// ---- 00_FunctionsBlocks/Beckhoff/DataProcessing/Database/SQLite_CreateDb_V2.TcPOU
PROGRAM SQLite_CreateDb_V2
VAR_INPUT
	IN_ConfigDbActuelle		: ARRAY[0..MAX_CONFIGURATIONS] OF ST_ConfigDB; 
	IN_DbType				: UINT:= 1; // 1:T_DBConfig_SQLite, 2:T_DBConfig_SQLCe
	IN_Dir					: T_MAXSTRING;
	IN_Name					: STRING;
	IN_Start				: BOOL;
	IN_TableName			: STRING;
END_VAR
VAR_IN_OUT
	IN_hDBID         		: UDINT;	
END_VAR
VAR_OUTPUT
	OUT_Error				: BOOL;
	OUT_Busy				: BOOL;
	OUT_Result				: INT;
END_VAR
VAR
	Etape					: UINT;
	
	TrigStart				: R_TRIG;
	RsStart					: RS;
	bCreateTable			: BOOL;
	TrigCreateTable			: R_TRIG;
	RsCreateTable			: RS;
	PLCDBCreateEvt 			: FB_PLCDBCreateEvt(sNetID := '', tTimeout := T#5S);
	SqlLiteConf				: T_DBConfig_SQLite;
	DbFullDirName			: T_MAXSTRING;	
	sExtension				: STRING:= '.db';
	tcMessage    	 		: I_TcMessage;
	
	AX_ColArray				: ARRAY[0..3] OF ST_ColumnInfo;
	
	dBID_Test				: UDINT;
	KK						: UDINT;
	bExisteDeja				: BOOL;	
END_VAR

OUT_Busy := TRUE;
AX_ColArray[0].sName := 'TimeStamp';     	AX_ColArray[0].eType := E_ColumnType.DateTime;   	AX_ColArray[0].nLength := 4;    
AX_ColArray[1].sName := 'TimeStamp_Ms';    	AX_ColArray[1].eType := E_ColumnType.Integer;    	AX_ColArray[1].nLength := 4;
AX_ColArray[2].sName := 'ParentId';   		AX_ColArray[2].eType := E_ColumnType.Integer;   	AX_ColArray[2].nLength := 4;
AX_ColArray[3].sName := 'Value';   			AX_ColArray[3].eType := E_ColumnType.Float;   		AX_ColArray[3].nLength := 8;


IF IN_DbType = 1 THEN
	sExtension := '.db';
ELSIF IN_DbType = 2 THEN
	sExtension := '.sdf';
END_IF

DbFullDirName := Concat(STR1:=Concat(STR1:= IN_Dir, STR2 := IN_Name), STR2 := sExtension);
SqlLiteConf.bAuthentification := FALSE;
SqlLiteConf.sServer := DbFullDirName;

FOR KK := 0 TO MAX_CONFIGURATIONS DO
	IF IN_ConfigDbActuelle[KK].sServer = DbFullDirName THEN
		bExisteDeja := TRUE;
		OUT_Result := -1;
		OUT_Busy := FALSE;
		OUT_Error := FALSE;
		bCreateTable := FALSE;
		IN_hDBID := IN_ConfigDbActuelle[KK].hDBID;
		EXIT;
	END_IF
	IF KK = MAX_CONFIGURATIONS THEN
		bExisteDeja := FALSE;
	END_IF
END_FOR

TrigStart(CLK := IN_Start AND NOT bExisteDeja);
RsStart(SET := TrigStart.Q);
IF RsStart.Q1 THEN
	IF PLCDBCreateEvt.Database(pDatabaseConfig := ADR(SqlLiteConf), cbDatabaseConfig := SIZEOF(SqlLiteConf), bCreateXMLConfig := TRUE, pDBID := ADR(dBID_Test)) THEN
		IF PLCDBCreateEvt.ipTcResult.nEventId = 59 THEN
			OUT_Error := FALSE;
			OUT_Result := -1;
			OUT_Busy := FALSE;	
			TrigStart(CLK := FALSE);
			bCreateTable := FALSE;
			Etape := 0;
			RsCreateTable(RESET1 := TRUE);
			RsCreateTable(RESET1 := FALSE);
		ELSIF PLCDBCreateEvt.bError THEN
			tcMessage := PLCDBCreateEvt.ipTcResult;
			OUT_Error := TRUE;
		ELSE
			Etape := 1;
			IN_hDBID := dBID_Test;
			bCreateTable := TRUE; 
		END_IF
		RsStart(RESET1 := TRUE);
		RsStart(RESET1 := FALSE);
	END_IF
END_IF

TrigCreateTable(CLK := bCreateTable);
RsCreateTable(SET:= TrigCreateTable.Q);

IF RsCreateTable.Q1 AND ETAPE = 1 THEN
	IF PLCDBCreateEvt.Table(hDBID := IN_hDBID, sTableName := IN_TableName,  pTableCfg := ADR(AX_ColArray), cbTableCfg := SIZEOF(AX_ColArray)  ) THEN
		IF PLCDBCreateEvt.bError THEN
			Etape := 255;
			OUT_Error := TRUE;
			OUT_Result := -2;
		ELSE
			IN_Start := FALSE;
			bCreateTable := FALSE;
			Etape := 0;
			OUT_Result := 1;
			RsCreateTable(RESET1 := TRUE);
			RsCreateTable(RESET1 := FALSE);
			TrigStart(CLK := False);
			OUT_Busy := FALSE;	
			OUT_Error := FALSE;
		END_IF
	END_IF
END_IF

IF Etape = 255 THEN
	Etape := 0;
	bCreateTable := FALSE;
	IN_Start := FALSE;
	OUT_Busy := FALSE;	
	RsCreateTable(RESET1 := TRUE);
	RsCreateTable(RESET1 := FALSE);
	
END_IF

END_PROGRAM

// ---- 00_FunctionsBlocks/Beckhoff/DataProcessing/Database/SQLite_DeleteConfDb.TcPOU
PROGRAM SQLite_DeleteConfDb
VAR_INPUT
	IN_DbType				: UINT:= 1; // 1:T_DBConfig_SQLite, 2:T_DBConfig_SQLCe
	IN_hDBID         		: UDINT;
	IN_Start				: BOOL;
	
END_VAR
VAR_OUTPUT
	OUT_Error				: BOOL;
	OUT_Busy				: BOOL;
END_VAR
VAR
	Etape					: UINT;
	
	TrigStart				: R_TRIG;
	RsStart					: RS;
	bDeleteTable			: BOOL;
	TrigDeleteFile			: R_TRIG;
	RsDeleteTable			: RS;
	fbConfigTcDBSrv   		: FB_ConfigTcDBSrvEvt (sNetID := '', tTimeout := T#5S);
	DbFullDirName			: T_MAXSTRING;	
	sExtension				: STRING:= '.db';
	tcMessage    	 		: I_TcMessage;
	
	

END_VAR

OUT_Busy := TRUE;

TrigStart(CLK := IN_Start);
RsStart(SET := TrigStart.Q);
IF RsStart.Q1 THEN
	IF fbConfigTcDBSrv.Delete(eTcDBSrvConfigType := E_TcDBSrvConfigType.Database, hConfigID := IN_hDBID) THEN
		IF fbConfigTcDBSrv.bError THEN
			tcMessage := fbConfigTcDBSrv.ipTcResult;
			OUT_Error := TRUE;
			OUT_Busy := FALSE;
			Etape := 255;
		ELSE 
			OUT_Busy := FALSE;
			OUT_Error := FALSE;
			Etape := 0;
		END_IF
		TrigStart(CLK := FALSE);
		RsStart(RESET1 := TRUE);
		RsStart(RESET1 := FALSE);
	END_IF
END_IF

IF Etape = 255 THEN
	Etape := 0;
	bDeleteTable := FALSE;
	IN_Start := FALSE;
	OUT_Busy := FALSE;	
	RsDeleteTable(RESET1 := TRUE);
	RsDeleteTable(RESET1 := FALSE);
	
END_IF

END_PROGRAM

// ---- 00_FunctionsBlocks/Beckhoff/DataProcessing/FB_MessageDynamique.TcPOU
FUNCTION_BLOCK FB_MessageDynamique
// Allows to create dynamic messages in order to add variable to a string
VAR_INPUT
	
	InMessage	: ST_ValuesAlarms;
	InNbparam	: SINT;
END_VAR
VAR_OUTPUT
	OutMessage	: STRING(150);
END_VAR
VAR
	Valeur  	: STRING(10); // Nom de la balise a tester
	P	    	: INT;		 // Pos de la balise dans une chaine de caractere 
	i,j			: SINT;		// Compteur incrémental
	Temp		: String(150);
END_VAR

Temp:=InMessage.Message;
FOR i:=1 TO InNbparam DO
	IF InMessage.Ax_ParamB[i]<>0 THEN
		Valeur := BOOL_TO_STRING(InMessage.Ax_ParamB[i]^);
		P      := FIND(Temp,concat('<Balise_B',INT_TO_STRING(i)));
		IF P >0 THEN
			Temp:=Replace(Temp,Valeur,10,P);
		ELSE
			EXIT;
		END_IF
	END_IF
END_FOR

FOR j:=1 TO InNbparam DO
	IF InMessage.Ax_ParamI[j]<>0 THEN
		Valeur := SINT_TO_STRING(InMessage.Ax_ParamI[j]^);
		P      := FIND(temp,concat('<Balise_I',INT_TO_STRING(j)));
		IF P >0 THEN
			Temp:=Replace(temp,Valeur,10,P);
		ELSE
			EXIT;
		END_IF
	END_IF
END_FOR
OutMessage:=Temp;

END_FUNCTION_BLOCK

// ---- 00_FunctionsBlocks/Beckhoff/DataProcessing/FUN_Transpose.TcPOU
PROGRAM FUN_Transpose
// Allows to transpose an array 
VAR_INPUT
	In_Array					: ARRAY[1..500] OF ARRAY[1..5] OF STRING;
END_VAR
VAR_OUTPUT
	Out_Array					: ARRAY[1..5] OF ARRAY[1..500] OF STRING;
END_VAR


VAR
	KK: INT;
	LL: INT;
END_VAR

FOR LL := 1 TO 5 DO 
	FOR KK := 1 TO 500 DO
	
		Out_Array[LL][KK] := In_Array[KK][LL];
		
	END_FOR
END_FOR

END_PROGRAM

// ---- 00_FunctionsBlocks/Beckhoff/DataProcessing/ReadFile/FB_ReadCSV.TcPOU
FUNCTION_BLOCK FB_ReadCSV
//Permet de lire les Valeurs de max 1 semaine de points (1 pt/min pdt 7 jours)

VAR_INPUT
	InDirectory_Stockage 		: T_MaxString;		// Base file of the Historization 
	InVariable					: T_MaxString;
	InStartTimeStamp			: TIMESTRUCT;
	InNbLecture					: UINT := 144;
	InExecute					: BOOL;			//Rising Edge detection of read
	ParamSeparateur				: STRING;
	InStructValues				: ARRAY[1..500] OF ST_ValuesWrite;
END_VAR                 		

VAR_OUTPUT              		
	OutValue					: ARRAY[1..10000] OF REAL;
	OutTimeStamp				: ARRAY[1..10000] OF TIMESTRUCT;
	OutCompleted				: BOOL;
	OutbBusy					: BOOL;
	OutError 					: BOOL;
	OutErrorID 					: UINT; // 1 : File not found
END_VAR                 		
VAR     
	// Initialisation 
	CP_READ						: BOOL;
	TypeFile					: STRING;
	ParamTimeOut				: TIME := T#1S;
	
	//Read
	TimeStructBeingRead			: TIMESTRUCT;
	FullDirectory				: STRING;                		
	ReadNewFile					: BOOL;
	
	
	OpenFile					: FB_FileOpen;
	ReadFile					: FB_FileGets;
	CloseFile					: FB_FileClose;
	LineStart					: UINT;			// Ligne de début de la lecture
	LineEnd						: UINT;			// Ligne de fin de la lecture
	LineLeft					: UINT;			// Nombre total de lignes restantes
	Index_Array_OutValue		: UINT;			// Valeur de OutValue qui va être écrite
	
	Opening						: BOOL := TRUE;
	Reading						: BOOL;
	Closing						: BOOL;
	LineRead					: ARRAY[1..20] OF T_Maxstring;
	LineReadNull				: ARRAY[1..20] OF T_Maxstring;
	ColumnNbRead				: UINT;
	TimeStampRead				: STRING(255);
	ValueRead					: STRING(255);
	EOF_Reached					: BOOL;
	PosCursor					: DINT;
                    		
	CompteurLigne				: CTU;
	CompteurLigneRead			: CTU;
	OutBusy						: RS;
	Trig_Read					: R_TRIG;
	Trig_Start 					: R_TRIG;
	
	FileHandle					: UINT;
	FileHandle_Old				: UINT;
	
	NbJours						: UINT;
	KK: UINT 					:= 1;
	bInit 						: BOOL;
	FinalElemStruct				: UINT := 20;
	LL							: UINT := 1;
	LenLineRead					: INT;
END_VAR

IF  Trig_Start.Q THEN
	M_Init();
END_IF

CP_Read := SYSTEMTIME_TO_DT(InStartTimeStamp) + LINT_TO_TIME(InNbLecture*60000) < SYSTEMTIME_TO_DT(CalLocalTimeStruct);
 Trig_Start(CLK := InExecute);
CompteurLigneRead(PV := InNbLecture, RESET := Trig_Start.Q);

OutBusy(Set := CP_Read AND InExecute, RESET1 := OutError OR OutCompleted);
OutbBusy := OutBusy.Q1;

OutCompleted := CompteurLigneRead.Q;

IF OutBusy.Q1 THEN	
	// J'initialise le tout : 
		//Initialisation du type de fichier
			TypeFile := 'RAWDATA'; 
			
		// Calcul du nb de fichiers à ouvrir
			NbJours := DINT_TO_UINT( TRUNC(UINT_TO_INT(InNbLecture + InStartTimeStamp.wHour *60 + InStartTimeStamp.wMinute)/(24*60))+1);

	IF KK <= NbJours THEN
		// Nbre d'heures * 60 + Nbre de minutes + 2 lignes de presentation
		IF KK = 1 THEN
			LineStart := (InStartTimeStamp.wHour *60 + InStartTimeStamp.wMinute + 2); 
			// Calcul des lignes de la lecture : 
			LineLeft := InNbLecture;
		ELSE
			LineStart := 2;
		END_IF
		
		LineEnd := MIN(1442, LineLeft);

		CompteurLigne(PV := LineStart+LineEnd);
		
		TimeStructBeingRead := DT_TO_SYSTEMTIME(SYSTEMTIME_TO_DT(InStartTimeStamp) + LINT_TO_TIME(24*3600000*(KK-1)));
		FullDirectory := Concat(Concat(Concat(Concat(Concat(Concat(Concat(Concat(Concat(Concat(Concat(Concat(InDirectory_Stockage , WORD_TO_STRING(TimeStructBeingRead.wyear)),'\'),WORD_TO_STRING(TimeStructBeingRead.wMonth)),'\'),'RAWDATA'),'_'),WORD_TO_STRING(TimeStructBeingRead.wyear)),'-'),WORD_TO_STRING(TimeStructBeingRead.wMonth)),'-'),WORD_TO_STRING(TimeStructBeingRead.wDay)),'.csv');

		//Ouverture du Fichier, récupération du handle
		OpenFile
		(
			sNetId := '',
			sPathName := FullDirectory,
			nMode := FOPEN_MODEREAD,
			ePath := PATH_GENERIC,
			bExecute := Opening AND NOT OutCompleted,
			hFile => FileHandle
		);
		
		IF OpenFile.nErrId = 1804 THEN // Le fichier n'existe pas 
			OutErrorID := 1;
			OutError := OpenFile.bError;
		ELSIF OpenFile.bError THEN		// Il y a eu une autre erreur
			OutError := OpenFile.bError;
		ELSIF NOT OpenFile.bError AND NOT OpenFile.bBusy AND FileHandle <> 0 AND FileHandle <> FileHandle_Old THEN
			Opening := FALSE;
			FileHandle_Old := FileHandle;
		END_IF
		// On a obtenu le file handle, on va commencer la lecture
		
		
		// Le bloc suivant va lire le document ligne à ligne en incrémentant le compteur ligne et en ressortant l'ensemble de la ligne dans LineRead
		
		IF NOT opening AND NOT CompteurLigneRead.Q AND NOT EOF_Reached THEN		
			IF LL <= 20 THEN
				ReadFile
				(
					sNetId := '',
					hFile := FileHandle,
					bExecute := TRUE,
					tTimeout := ParamTimeOut,
					sLine => LineRead[LL],
					bEOF => EOF_Reached
				);	
				IF NOT ReadFile.bBusy AND NOT ReadFile.bError AND lineread[LL] <> '' THEN
					ReadFile(bExecute := FALSE);
					LenLineRead := LEN(STR := LineRead[LL]);
					IF LenLineRead = 254 THEN
						LL := LL + 1 ;
					ELSE
						FinalElemStruct := LL;
						LL := 1;
					END_IF
				END_IF
			END_IF
			
			IF NOT ReadFile.bBusy AND NOT ReadFile.bError AND (LineRead[FinalElemStruct] <> '' OR EOF_Reached) THEN
				ReadFile(bExecute := FALSE);
				CompteurLigne(CU := TRUE);	
				CompteurLigne(CU := FALSE);
				FinalElemStruct := 20;
				
				IF CompteurLigne.CV >= LineStart + 1 THEN
					TimeStampRead := Substring_Cari
					(
						IN_Delimiter := ParamSeparateur, 
						IN_TextToSearch := LineRead, 
						IN_Position := 0
					);
					OutTimeStamp[Index_Array_OutValue+1]:= FUN_FormatDate(In_String := TimeStampRead);
					
					ValueRead := Substring_Cari
					(
						IN_Delimiter := ParamSeparateur, 
						IN_TextToSearch := LineRead, 
						IN_Position := ColumnNbRead + 1
					);
					OutValue[Index_Array_OutValue+1] := STRING_TO_REAL(ValueRead)*100;
					CompteurLigneRead(CU := TRUE);
					CompteurLigneRead(CU := FALSE);
					Index_Array_OutValue := Index_Array_OutValue + 1;
					
					LL := 1;
				END_IF
				LineRead := LineReadNull;
			ELSIF NOT ReadFile.bBusy AND  ReadFile.bError THEN
				OutError := TRUE;			
			END_IF
		ELSIF EOF_Reached THEN
			ReadFile(bExecute := FALSE);
	
			CloseFile
			(
				sNetId := '',
				bExecute := TRUE,
				hFile := FileHandle,
				tTimeout := ParamTimeOut
			);
			IF NOT CloseFile.bBusy AND NOT CloseFile.bError  THEN
				LineLeft := LineLeft - CompteurLigneRead.CV + 2;
				Index_Array_OutValue := Index_Array_OutValue -1;
				CloseFile(bExecute := FALSE);
				CompteurLigne(RESET := TRUE);
				CompteurLigne(RESET := FALSE);
				Opening := TRUE;
				EOF_Reached := FALSE;
				KK := KK + 1;
			END_IF	
		END_IF
	END_IF
ELSIF EOF_Reached OR CompteurLigneRead.Q AND FileHandle <> 0 THEN
	ReadFile(bExecute := FALSE);
	
	CloseFile
	(
		sNetId := '',
		bExecute := TRUE,
		hFile := FileHandle,
		tTimeout := ParamTimeOut
	);
	IF NOT CloseFile.bBusy AND NOT CloseFile.bError THEN
		CloseFile(bExecute := FALSE);
		CompteurLigne(RESET := TRUE);
		CompteurLigne(RESET := FALSE);
		Opening := TRUE;
		Index_Array_OutValue := 0;
		FileHandle := 0;
		KK := 1;
	ELSIF NOT CloseFile.bBusy AND closefile.bError THEN
		OutError := TRUE;
	END_IF  
END_IF

METHOD M_Init : BOOL
VAR_INPUT
END_VAR

VAR
	KK : UINT;
END_VAR
ColumnNbRead := 1;
FOR KK := 1 TO 500 DO
	IF InVariable = InStructValues[KK].Description THEN
		ColumnNbRead := KK;
		EXIT;
	END_IF
END_FOR
END_METHOD

END_FUNCTION_BLOCK

// ---- 00_FunctionsBlocks/Beckhoff/DataProcessing/WriteFile/CheckStruct_Alarms.TcPOU
FUNCTION CheckStruct_Alarms : BOOL
//Allows to compare 2 Struct_InputRTU, TRUE if struct are the same
VAR_INPUT
	InStruct1 : ST_ValuesAlarms;
	InStruct2 : ST_ValuesAlarms;
END_VAR
VAR
	bCompareBuffer 	: BOOL := TRUE;
	KK 				: UINT;
END_VAR

CheckStruct_Alarms := InStruct1.Message = Instruct1.Message and InStruct1.ID = Instruct2.ID and InStruct1.Value = InStruct2.Value and InStruct1.Written = Instruct2.Written;

END_FUNCTION

// ---- 00_FunctionsBlocks/Beckhoff/Fifo/FB_CommandAlternate.TcPOU
FUNCTION_BLOCK FB_CommandAlternate
VAR_INPUT
	AX_CMD 			: ARRAY[1..6] OF INV_Cmd;
	In_NB_Prio		: UINT;							
	ParamNbCMD		: UINT := 6;					// Number of elements of AX_CMD array
	In_Pulse		: BOOL;
END_VAR

VAR_OUTPUT
	CmdOutput		: INV_Cmd	;
END_VAR
VAR
	LastPosition 	: UINT;
	KK				: UINT;
	bInterrupt		: BOOL;
	Debut			: UINT;
	Fin				: UINT;
	Trig_Detec		: R_TRIG;
END_VAR

bInterrupt := FALSE;
Trig_Detec(CLK := In_Pulse);

IF Trig_Detec.Q THEN
	FOR KK := 1 TO In_NB_Prio DO
		IF AX_CMD[KK].bCmdStart^ THEN
			bInterrupt 	:= TRUE;
			CmdOutput := AX_CMD[KK];
			EXIT;
		END_IF
	END_FOR
	
	IF NOT bInterrupt THEN
		Debut := MAX(In_NB_Prio + 1, LastPosition + 1);
		Fin := Debut + ParamNbCMD - In_NB_Prio - 1;
		FOR KK := Debut TO Fin DO
			IF AX_CMD[KK - BOOL_TO_UINT(KK > ParamNbCMD)*(Fin - Debut + 1)].bCmdStart^ THEN
				LastPosition := KK - BOOL_TO_UINT(KK > ParamNbCMD)*(Fin - Debut + 1);
				CmdOutput := AX_CMD[ KK - BOOL_TO_UINT(KK > ParamNbCMD)*(Fin - Debut + 1)];
				EXIT ;
			END_IF
		END_FOR
	END_IF
END_IF

END_FUNCTION_BLOCK

// ---- 00_FunctionsBlocks/Common/AlarmManagement/FB_DetectFixedValue.TcPOU
FUNCTION_BLOCK FB_DetectFixedValue
VAR_INPUT
	IN_Addr			: POINTER TO BYTE;			// Adr of the variable to  analyse
	IN_EmptyStruct	: POINTER TO BYTE;			// Adr of a null variable on which I input the compared value
	IN_Size			: UINT;						// Size of the variable to analyse
	IN_Duration		: TIME;						// Duration after which an alarm is raised
END_VAR
VAR_OUTPUT
	OUT_bStatic		: BOOL;						// Value has been static for more than IN_Duration time
END_VAR
VAR
	TON_CMP			: TON;
	bFixed			: BOOL;
END_VAR

bFixed :=  MEMCMP(pBuf1 := IN_Addr, pBuf2 := IN_EmptyStruct, n := IN_SIZE)=0;

TON_CMP(IN := bFixed, PT := IN_Duration, Q => OUT_bStatic);

IF NOT bFixed THEN
	MEMCPY(destAddr := IN_EmptyStruct, srcAddr := IN_Addr, n := IN_Size);
END_IF

END_FUNCTION_BLOCK

// ---- 00_FunctionsBlocks/Common/AlarmManagement/FB_UnknownEvent.TcPOU
FUNCTION_BLOCK FB_UnknownEvent
////////////////// 
// Detect an event that is not the result of an internal command, or an external event
//////////////////	
VAR_INPUT
	IN_TempoAfterCommand					: TIME ;					// Tempo between internal command and event
	IN_TempoReadExternalEvent					: TIME ;					// Tempo to read the external event
	
	IN_InternalCommand				: BOOL ; 			// Internal command that normally trigers the event 
	IN_ExternalEvent				: BOOL ; 			// External Event that normally explains the Event (to be read after the event)
	
	IN_Event						: BOOL ; // Event that occur
	
	bReset				: BOOL := FALSE ; 	// Reset 
	
END_VAR

VAR_OUTPUT
	OUT_Unknown 			: BOOL ; 		// Flag to TRUE is the event is unknown ( neither related to the command, or an external event that is known) 
	
END_VAR

VAR
	FB_CheckCommand : FB_CheckCommand ;
	// Inconsistency detection
	R_TRIG1				: R_TRIG ; 		// Detect command
	TOF1				: TOF ; 		// Creates a falling edge T time after command detcetion	
	F_TRIG				: F_TRIG ; 		// Detect Falling edge of TOF1	
	
	F_TRIG2				: F_TRIG ; 		// Detect falling edge of feedback measure
	TOF2				: TOF ; 		// Creates  a falling edge T time after Feedback measure ended detcetion
 
	TON					: TON ; 		// Tempo in case of bistable functuion

	// Reset management 	
	TOF_Reset			: TOF;			// Hold Reset command afetr reset to inhibate future warnings
	RS_Reset			: RS;			// Maintain reset command
	
	R_TRIG2: R_TRIG;
	CalNotLinkedToCommand: BOOL;
END_VAR


R_TRIG1(CLK := IN_InternalCommand) ; 

TOF1(IN:=R_TRIG1.Q , PT:=IN_TempoAfterCommand) ;
F_TRIG(CLK:=TOF1.Q);		

R_TRIG2(CLK := IN_Event) ; 


CalNotLinkedToCommand :=  NOT TOF1.Q AND R_TRIG2.Q ;
 
FB_CheckCommand(T:= IN_TempoReadExternalEvent , bCmd := CalNotLinkedToCommand , bMes := IN_ExternalEvent , bReset := bReset , bImpulsion := TRUE ) ; 
OUT_Unknown := FB_CheckCommAND.bWarning  ;

END_FUNCTION_BLOCK

// ---- 00_FunctionsBlocks/Common/BoolManagement/FB_CountNinTimeWindow.TcPOU
FUNCTION_BLOCK FB_CountNinTimeWindow
VAR_INPUT
	IN_CountMax			: UINT := 3 ; 
	IN_bInput				: BOOL;
	IN_bReset			: BOOL;
END_VAR
VAR_OUTPUT
	OUT_FlagNinT		: BOOL;		// Output : if CountMax Input occured in the last T min, this variable = TRUE;
END_VAR
VAR
	TimeFault1			: TIME;		// Temps du troisième défaut GTE (chronologiquement parlant)
	TimeFault2			: TIME;		// Temps du deuxième défaut GTE (chronologiquement parlant)
	TimeFault3			: TIME;		// Temps du premier défaut GTE (chronologiquement parlant)
	TriggerGTE			: R_TRIG;	
	
	TestDiff			: TIME;
END_VAR
VAR_INPUT PERSISTENT
	ParamTimeToMeasure	: TIME := T#30M; // Time during which the 3 GTE are measured. Used for testing.
END_VAR

TriggerGTE(CLK:= IN_bInput);

 IF IN_bReset THEN
		OUT_FlagNinT := FALSE;
		TimeFault1 := T#0S;
		TimeFault2 := T#0S;
		TimeFault3 := T#0S;
END_IF

IF TriggerGTE.Q AND TimeFault3 = T#0S THEN
	TimeFault3 := TIME();
ELSIF TriggerGTE.Q AND TimeFault2 = T#0S THEN
	TimeFault2 := TIME();
ELSIF TriggerGTE.Q AND TimeFault1 = T#0S THEN
	TimeFault1 := TIME();
ELSIF TriggerGTE.Q THEN
	TimeFault3 := TimeFault2;
	TimeFault2 := TimeFault1;
	TImeFault1 := TIME();
END_IF


IF TimeFault1 - TimeFault3 < ParamTimeToMeasure AND TimeFault1 <> T#0S THEN
	OUT_FlagNinT := TRUE;
ELSE 
	OUT_FlagNinT := FALSE;
END_IF

END_FUNCTION_BLOCK

// ---- 00_FunctionsBlocks/Common/BoolManagement/FB_Toggle2Tap.TcPOU
FUNCTION_BLOCK FB_Toggle2Tap
///////////
// FB to change a toggle into a tap with constant duration//
///////////

VAR_INPUT
	TapDuration		: TIME; 	// (s) Tap duration
	
	ToggleVar 		: BOOL;		// Toggled input variable 

	
END_VAR

VAR_OUTPUT
	TapVar			: BOOL ; 	// Tapped output variable
	
END_VAR

VAR				
	R_TRIG			: R_TRIG ;				// Create a square at Rising Edge Detection
	F_TRIG			: F_TRIG ;				// Create a square at falling Edge Detection 
	TP				: TP ; 					// Square Signal 

END_VAR

R_TRIG(CLK := ToggleVar) ;  							// Rising Edge Detection
F_TRIG(CLK := ToggleVar) ; 								// Falling Edge Detection

TP(IN := R_TRIG.Q OR F_TRIG.Q , PT := TapDuration) ;  	// Square signal 

TapVar		:= TP.Q ; 									// OUtput variable

END_FUNCTION_BLOCK

// ---- 00_FunctionsBlocks/Common/BoolManagement/FB_WriteOnChange.TcPOU
FUNCTION_BLOCK FB_WriteOnChange
////////////////// 
// Write output variable , equals to input variable only if input variable changed state 
//////////////////	

VAR_INPUT
	Size			: UDINT; 				// Variable size 
	VarOut			: POINTER TO BYTE;		// Output  Variable Memory Address
	VarInput		: POINTER TO BYTE;		// Input Variable Memory Address	
END_VAR


VAR
	VarHold 		: DWORD  ; 	

END_VAR

IF MEMCMP(pBuf1:= VarInput, pBuf2:= ADR(VarHold) , n:=Size )<>0  THEN
	MEMCPY(srcAddr:= VarInput , destAddr := VarOut, n:= Size ) ;
END_IF

IF MEMCMP(pBuf1:= VarOut, pBuf2:= ADR(VarHold) , n:=Size )<>0  THEN
	MEMCPY(srcAddr:= VarOut , destAddr := VarInput, n:= Size ) ;
END_IF

MEMCPY(srcAddr:= VarInput , destAddr := ADR(VarHold), n:= Size ) ;

END_FUNCTION_BLOCK

// ---- 00_FunctionsBlocks/Common/BoolManagement/RS_NoReset.TcPOU
FUNCTION_BLOCK RS_NoReset
//Output reset the input if the input is false 
VAR_INPUT
	Set 		: BOOL;
	Reset 		: BOOL;
END_VAR
VAR_OUTPUT
	Q1 			: BOOL;
END_VAR
VAR
	TRIG 		: R_TRIG;
	RS 			: RS;
END_VAR

TRIG(CLK := Set);
RS(Set := TRIG.Q, RESET1 := Reset AND NOT Set, Q1 => Q1);

END_FUNCTION_BLOCK

// ---- 00_FunctionsBlocks/Common/Ctrl/FB_PIDRegulation.TcPOU
FUNCTION_BLOCK FB_PIDRegulation
// Akuo Version of PID Regulation  for solar power plant . Input can be P or Q . 
// Out  = Error *K (1+ 1/Ti sum(error) + Td delta(error) ) 
(*
	DATE :						07/2020																										
	Developper:				GGY																												
	Version :					V1.0																										
	Function :																																																																		
*)
VAR_INPUT PERSISTENT

	ParamK				: REAL ; // Proportionnal 
	ParamTi				: REAL ; // Integral (s) . 0 to disable
	ParamTd				: REAL ; // Derivative (s). 0 to disable . 
	
	ParamXmax			: REAL ; // maximal Value for X. Shall account for number of available PTR . 
	ParamXmin			: REAL; // minimal value for X 
	
	ParamOutmax			: REAL ; // Maximal output value
	ParamOutmin			: REAL ; // Maximal input value 
	
	
	
END_VAR

VAR_INPUT
	IN_SetptX				: REAL ; // Value to reach 
	IN_MesX					: REAL ; // Measure to compare with
	IN_MesComXError			: BOOL ; // Communication lost with the measure tool. 
	IN_SetptOpenLoop		: REAL  ; // Output of the PID when disabled. This shall be equal to an evaluation of the correct output. Usually SetptX. OpenLoop setpoint. 

	
	IN_CmdReset				: BOOL ; // Reset PID 
	IN_CmdPIDOn				: BOOL ; // Activate/ Desactivate PID . outpout equals to the offset if desactivated/ 
END_VAR

VAR_OUTPUT
	OUT_X					: REAL ; // Output of the PID 
	OUT_PIDMode				: INT ; // Mode of the PID ( 1: Bypassed  , 3 : Proportionnal , 4 : PI , 5 PID , 6: PD). 
	
END_VAR
VAR
	
	CalSetptOffset 			: REAL  ; // Offset to be added to the PID to ensure continuity when resetting it or activating it. 

	IntegralX			: REAL ; // Intergal
	DerivativeX			: REAL ; // Derivative
	ErrorX				: REAL;	// Error  
	CP_PID				: BOOL;	// PID Enabled
	Clock				: TON ; // Calculate Elapsed Time ; 
	DeltaTime			: REAL ; // 
	// Derivative
	StepDerivative		: INT := 0; // Derivative Step ( initialization , methode degre 1 , methode degre 2) 
	X2,X1				:REAL;
	T1					:REAL;
	CalReset: BOOL;
	
	KCopy				: REAL ; 
	TiCopy				: REAL ; 
	TdCopy				: REAL ; 
	X_Temp				: REAL ; // Intermediate result . 
	
	CalOutLimitReached_Up	: BOOL;		// Output reached maximum output limit
	CalOutLimitReached_Down	: BOOL;		// Output reached minimum output limit
	
	TrigCP_PID: BOOL;
	bInit: BOOL := TRUE  ; 
	time_new: INT;
	delta_time: INT;
	time_old: INT;
END_VAR

// INITIALIZE 
	OUT_PIDMode := 1 ;

	CalReset := IN_CmdReset OR NOT IN_CmdPIDOn OR ABS(KCopy-ParamK)>0.000001 OR ABS(TiCopy-ParamTi)>0.000001 OR ABS(TdCopy-ParamTd)>0.000001 OR IN_MesComXError; // Reset if change of parameters >> passage en boucle ouverte. 

	CP_PID :=   (ParamK>0.00001 OR ParamK<-0.00001)  AND NOT CalReset  ; // PID Enable ssi Activation and K >0 and not communication alarm with power meter . and not K change . 
	

	IF NOT CP_PID OR bInit THEN 
		// Début proposition de modif KBT
		time_old := TIME_TO_INT(TIME());
		// Fin proposition de modif KBT

		
		Clock(IN:=FALSE ) ; 
		Clock(IN:=TRUE, PT:=T#1H);	//Initialize clock 
		bInit	:= FALSE ; 
	ELSE 
		Clock();
		DeltaTime	:= TIME_TO_REAL(CLOCK.ET)/1000 ; 	// in seconds
		
		// Début proposition de modif KBT
		time_new := TIME_TO_INT(TIME());
		IF time_old <> 0 THEN
			delta_time := time_new - time_old;
		END_IF
		time_old := TIME_TO_INT(TIME());
		// Fin proposition de modif KBT
	END_IF


	KCopy 	:=  ParamK ; 
	TiCopy	:= ParamTi ; 
	TdCopy	:= ParamTd ; 
	
// CHECK INPUT // 
	IN_SetptX := MAX(MIN(IN_SetptX, ParamXmax ), ParamXmin); // Limit the Input with Min/ Max values.

	IN_SetptOpenLoop := MAX(MIN(IN_SetptOpenLoop, ParamXmax ), ParamXmin); // Limit the Input with Min/ Max values.
	
// EVALUATE QUANTITIES //
	// Clock
	
	IF DeltaTime > 0 THEN	// We calculate on time cycle. When the time cycle is over , we reinitialize the clock
		Clock(IN:=FALSE ) ; 
		Clock(IN:=TRUE, PT:=T#1H);	//Initialize clock 
	ELSE
		CLOCK(PT:=T#1H,IN:=TRUE);
	END_IF
	// Error 
		ErrorX := IN_SetptX - IN_MesX ; 

	//Integral
		// Sauturate the integral if overflow or if limts are reached or output reaches limits Reset the integral if command reset. 
		IF (NOT(1E30 - ErrorX*DeltaTime < IntegralX OR -1E30 - ErrorX*DeltaTime > IntegralX) AND ParamTi>0 ) OR CalReset THEN
			IF NOT ((ErrorX > 0 AND  CalOutLimitReached_Up) OR (ErrorX < 0 AND CalOutLimitReached_Down)) THEN 
				IntegralX:=SEL(CalReset,IntegralX+ErrorX*DeltaTime , 0) ;
			END_IF
			
			
		END_IF
		
	// Derivative 
		IF StepDerivative=0 OR CalReset THEN		// Reinitializa derivative if reset commAND  
			X1:=ErrorX;
			X2:=ErrorX;
			T1:=DeltaTime;
			DerivativeX := 0;
			StepDerivative:=1;
		ELSIF StepDerivative=1 AND ParamTd>0 THEN 
			DerivativeX := (ErrorX - X1)/(DeltaTime-T1) ; // f'(x) = (f(x+h)-f(x))/h
			X2:=X1;
			X1:=ErrorX;
			T1:=DeltaTime;	
			StepDerivative:=2 ; 		
		ELSE	
			IF DeltaTime>0 AND DerivativeX < 1E30 AND ParamTd>0  THEN		// Saturate the derivative if going too high. 
				IF NOT ((ErrorX > 0 AND  CalOutLimitReached_Up) OR (ErrorX < 0 AND CalOutLimitReached_Down)) THEN  
					DerivativeX:=(3*(ErrorX)-4*X1+X2)/(2*(DeltaTime-T1));		// Formule de Gear au second degré décentré à gauche . f'(x) = 1/2h*(3*f(x+2h)-4*f(x+h)+f(x))  >>> https://www.imo.universite-paris-saclay.fr/~francois.dubois/cours/iacs/iacs-chap05.pdf
					X2:=X1;
					X1:=ErrorX;
					T1:=DeltaTime;
				END_IF
			END_IF;
		END_IF;
	
// PID CALCULATION
	IF CP_PID THEN

		
		TrigCP_PID	:= TRUE ; 
		// PID Enable 
		IF  ParamTi>0 AND ParamTd>0 THEN // Integral and derivative activated
			X_Temp:=CalSetptOffset+ParamK*(ErrorX+IntegralX/ParamTi+DerivativeX*ParamTd);
			OUT_PIDMode := 5 ; 
		ELSIF ParamTd>0 THEN // Derivative activated 
			X_Temp:= CalSetptOffset+ParamK*(ErrorX+DerivativeX*ParamTd) ; 
			OUT_PIDMode := 6 ; 
		ELSIF ParamTi>0 THEN // Integral activated 
			X_Temp:=CalSetptOffset+ParamK*(ErrorX+IntegralX/ParamTi);
			OUT_PIDMode := 4 ; 
		ELSE	// Only proportionnal
			X_Temp:=CalSetptOffset+ParamK*(ErrorX) ; 
			OUT_PIDMode := 3 ; 
		END_IF
		
	ELSE
		
		CalSetptOffset := IN_SetptOpenLoop ; // At the moment when i activated the PID, i need to ensure continuity of the OUT_X and start the PID from there . 
	
		TrigCP_PID	:= FALSE ; 
		//PID Disable. Open Loop . 
		X_Temp := IN_SetptOpenLoop ;
		OUT_PIDMode:=1 ;
	END_IF
	
// Saturate the OUtput with limits : 
CalOutLimitReached_Up := (X_Temp > ParamOutmax)  ;
CalOutLimitReached_Down:= (X_Temp < ParamOutmin)  ;
 

OUT_X :=  MAX(MIN(ParamOutmax , X_Temp ) , ParamOutmin ) ;

END_FUNCTION_BLOCK

// ---- 00_FunctionsBlocks/Common/DataProcessing/FB_CountBitOfWordAtTrue.TcPOU
FUNCTION_BLOCK FB_CountBitOfWordAtTrue
// Count the number of active bit of a word
VAR_INPUT
	MyWord		 	: WORD;		
END_VAR
VAR_OUTPUT
	NbrBitAtTrue 	: BYTE;
	PosOfLastOne	: BYTE;
END_VAR
VAR
	KK 			 	: BYTE;
	VarTemp		 	: WORD;
END_VAR


NbrBitAtTrue := 0;
FOR KK := 1 TO 16 DO
	Vartemp := ROL(MyWord, KK);
	IF VARtemp.0 THEN
		NbrBitAtTrue := NbrBitAtTrue +1 ;
		PosOfLastOne := KK;
	END_IF
END_FOR

END_FUNCTION_BLOCK

// ---- 00_FunctionsBlocks/Common/DataProcessing/FB_Integrate.TcPOU
FUNCTION_BLOCK FB_Integrate
// This FB increments the value of the Input with every call of the FB. DO NOT CALL THIS TWICE IN A CYCLE.
// Integration is done with the trapeze method
// The Reset input resets the value to 0
VAR_INPUT
	IN_DataToIntegrate		: REAL;
	IN_CmdReset				: BOOL;
	
END_VAR
VAR_OUTPUT
	OUT_IntegrationValue	: REAL;
END_VAR
VAR
	OldData					: REAL;
	OldTime					: TIME;
	DeltaTime				: TIME;
END_VAR

IF OldTime > T#0S THEN
	DeltaTime := TIME()-OldTime;
	
	OUT_IntegrationValue := OUT_IntegrationValue+(IN_DataToIntegrate + OldData)*TIME_TO_REAL(DeltaTime)/2000.0;
	
	OldTime := TIME();
	OldData := IN_DataToIntegrate;
	
	IF IN_CmdReset THEN
		OUT_IntegrationValue := 0.0;
		OldData := 0.0;
	END_IF
ELSE
	OldTime := TIME();
	OldData := IN_DataToIntegrate;
END_IF

END_FUNCTION_BLOCK

// ---- 00_FunctionsBlocks/Common/DataProcessing/FB_MovingAverage.TcPOU
FUNCTION_BLOCK  FB_MovingAverage
//////////////////
// Calculate the Moving Average of a data. Maximal number of point.
//////////////////

VAR CONSTANT 
	CstNbPointMax			: INT := 1000 ; // Average on one hour, with seconds granularity points

END_VAR


VAR_INPUT
	WindowDuration		: DINT ; // (ms) Window of Time during which the average will be done . 
	ValueIn 			: REAL ; // Value to average
	UpdatePeriod		: DINT ; // (ms) Period at which the value is updated. 	
	CycleTime			: INT := CstCycleTime_G; // (ms) Cycle time of the CPU
END_VAR
	

VAR_OUTPUT
	ValueOut			: REAL ; // Averaged Value. 
	bError 				: BOOL ; // Switch to true if error i inputs				
END_VAR

VAR
	Values 				: ARRAY[1..CstNbPointMax] OF REAL; 	// Value to remove from the average calculation
	
	NbPoints			: DINT ; 	// Number of points used for calculating the average. 
	PointPickUpNb		: DINT ; 	// Number of points to skip in average calculation
	
	JJ					: DINT;		// Pick Up index . 
	KK					: DINT;		// For Loop 
	
END_VAR

// EVALUATE VARIABLES //
PointPickUpNb 	:= UpdatePeriod		/	CycleTime ;
NbPoints 		:= WindowDuration 	/ 	UpdatePeriod  ;  

// CHECK INPUTS //
IF NbPoints > CstNbPointMax THEN 
	bError 		:= TRUE ; 
	ValueOut 	:= -1 ;
	
ELSE
	// UPDATE VALUE ARRAY WITH NEW VALUE AND REMOVE OLD ONE //
	JJ			:=JJ+1 ;
	
	IF JJ = PointPickUpNb THEN 
		JJ		:= 0 ; // Reinitialize JJ
		
		// Move all values in the array on the right
		FOR KK :=1 TO NbPoints-1 DO 
			Values[NbPoints-KK+1]	:= Values[NbPoints-KK] ;
			
		END_FOR
		
		Values[1] 					:= ValueIn ; 	// Assign first index to new value. 
		
		// CALCULATE AVERAGE // 
			ValueOut 						:= 0 ; 
			
			FOR KK:=1 TO NbPoints DO 
				ValueOut 					:= ValueOut + Values[KK] / DINT_TO_REAL(NbPoints) ; 
			
			END_FOR
		
	END_IF
END_IF

END_FUNCTION_BLOCK

// ---- 00_FunctionsBlocks/Common/DataProcessing/FB_Ramp.TcPOU
FUNCTION_BLOCK FB_Ramp
VAR_INPUT
	IN			: REAL;							(* New Setpoint variable *)
	ASCEND		: REAL;					(* maximum positive slope. Set negative value for no limit *)
	
	DESCEND		: REAL;				(* maximum negative slope (non-negative!!).Set negative value for no limit *)
	TIMEBASE	: TIME;					(* reference for ASCEND/DESCEND :
											t#0s : ASCEND/DESCEND defined per call
											else : ASCEND/DESCEND defined per specified time *)
	IN_RESET_VALUE		: REAL; // Value at which the OUT is reseted 
	RESET				:BOOL;						(* reset *)
END_VAR
VAR_OUTPUT
	OUT								: REAL;						(* output limited by  slope *)
	Out_Completed 					: BOOL ; // True when the ramp is over. 
END_VAR
VAR
	DIFF: REAL;
	OLD_IN: REAL;
	TB,CET:DWORD;
	CLOCK: TON;
	probe:REAL;
END_VAR

Out_Completed := FALSE ;

IF RESET=TRUE OR CLOCK.PT<>TIMEBASE THEN			(* Reset *)
	OUT :=  IN_RESET_VALUE ; 
	OLD_IN:=OUT;
	CLOCK(PT:=TIMEBASE,IN:=FALSE);
	Out_Completed := TRUE  ;
END_IF

DIFF:=IN-OLD_IN;									(* Calculate setpoint difference between old and new setpoint *)

IF TIMEBASE=T#0S THEN								(* PLC Cycletime *)
	IF DIFF>ASCEND AND ASCEND >0 THEN
		OUT:=OLD_IN+ASCEND;
	ELSIF DIFF<-DESCEND AND DESCEND >0 THEN
		OUT:=OLD_IN-DESCEND;
	ELSE
		OUT:=IN;
		Out_Completed := TRUE  ;					// 
	END_IF;
ELSE												(* Slope per timebase *)
	TB:=TIME_TO_DWORD(TIMEBASE);					(* TIMEBASE as DWORD *)
		CLOCK();
	CET:=TIME_TO_DWORD(CLOCK.ET);					(* Elapsed time : correspond to cycle time*)
	IF CET>0 THEN									(* *)
		CLOCK(IN:=FALSE);							(* Restart timer *)
		CLOCK(IN:=TRUE);
		probe:=DIFF*TB/CET;							// SMesIng value difference to fit timebase
		IF probe>ASCEND AND ASCEND >0 THEN						(* ascending *)
			OUT:=OLD_IN+ASCEND*CET/DWORD_TO_REAL(TB);
		ELSIF probe<-DESCEND AND DESCEND >0 THEN					(* descending *)
			OUT:=OLD_IN-DESCEND*CET/DWORD_TO_REAL(TB);
		ELSE										(* If value between max descend and max ascend.  *)
			OUT:=IN;
			Out_Completed := TRUE  ;
		END_IF;
	ELSE											(* keine Zeit verstrichen *)
		CLOCK.PT:=TIMEBASE;							(* => ggf. Initialisierung *)
		CLOCK(IN:=TRUE);							(* => ggf. Timer neu starten *)
		Out_Completed := TRUE  ;
	END_IF;
END_IF;

OLD_IN:=OUT;

END_FUNCTION_BLOCK

// ---- 00_FunctionsBlocks/Common/DataProcessing/FB_Ramp_Time.TcPOU
FUNCTION_BLOCK FB_Ramp_Time
// Y := Ax + B while bStart is set
// Works with time : You can set a max time, and a duration of the ramp :
// if pause is True, the Y value freezes until pause goes to False
// if max time is reached, the Y value goes to the value at maxtime

VAR_INPUT
	A 								: REAL ;	// Slope of the ramp
	B 								: REAL ;	// Initial value of the ramp
	bStart 							: BOOL ;	// Rising edge detection to start the ramp, if false, the ramp stops
	bPause							: BOOL ; 	// Pause signal : the value stop, then continues when bPause goes to false
	RampTime						: TIME ;	// Duration of the ramp
	MaxRampTime						: TIME ; 	// Maximum duration of the ramp (including breaks)
END_VAR                 			

VAR_OUTPUT              			
	Y 								: REAL;
	OutCompleted					: BOOL; 	// Rising edge detection to indicate the ramp is done
END_VAR                 		
	
VAR                     			
	TimeStart 						: TIME;
	TimeDurationPause 				: TIME;
	TimeOnGoing						: TIME;
	TimePauseold					: TIME;
	
	Trig_Start						: R_TRIG;
	Trig_Stop						: F_TRIG;
	Trig_PauseStart					: R_TRIG;
    Trig_OutCompleted				: R_TRIG;
            			
	Real_TimeSinceInit 				: REAL;
	                    	
	RS_TimerOn						: RS;
	TP_RampMaxTime					: TP;
END_VAR

Trig_Start(CLK := bStart);
TP_RampMaxTime(IN := Trig_Start.Q, PT := MaxRampTime);


//Trig_Stop(Clk := bStart AND TP_RampMaxTime.Q );
Trig_PauseStart(CLK := bPause);
Trig_OutCompleted(CLK := RS_TimerOn.Q1 AND TimeOnGoing = RampTime);

RS_TimerOn(SET := Trig_Start.Q, RESET1 := TimeOnGoing = RampTime OR Trig_Stop.Q OR Trig_OutCompleted.Q);


OutCompleted := Trig_OutCompleted.Q;
IF Trig_Start.Q THEN
	TimeStart := TIME();
	TimeDurationPause := T#0S;
	TimePauseOld := T#0S;
END_IF

IF Trig_PauseStart.Q THEN
	TimePauseOld := TIME();
END_IF

IF Trig_OutCompleted.Q THEN
	Trig_OutCompleted(CLK := FALSE);
	TimeOnGoing := T#0S;
END_IF

IF bPause THEN
	TimeDurationPause := TimeDurationPause + TIME() - TimePauseOld;
	TimePauseOld := TIME();
END_IF

IF RS_TimerOn.Q1 THEN
	TimeOnGoing := TIME() - TimeStart - TimeDurationPause;
	Real_TimeSinceInit := TIME_TO_REAL(TimeOnGoing);
	IF TimeStart > T#0S THEN
		Y := B + A * (Real_TimeSinceInit);
	END_IF
END_IF

END_FUNCTION_BLOCK

// ---- 00_FunctionsBlocks/Common/DataProcessing/FB_Smooth.TcPOU
FUNCTION_BLOCK FB_Smooth
////////////////// 
// Smooth Variable Change.
//////////////////	

VAR_INPUT
	Setpoint 		: REAL	:=0.0; 		// Setpoint variable
	Slope 			: REAL	:=5.0; 		// Slope in % of Range per seconds
	DeadBand 		: REAL 	:=2; 		// Deadband in % of Range
	Range 			: REAL; 			// Scale in which the value can evolve 
	CycleTime 		: REAL 	:= 1.0 ; 	// Cycle Time in ms.
	InitialValue 	: REAL ; 			// Initial Value of Slope after Reset
	
	Reset 			: BOOL ; 			// Reset initial Value at rising edge
	
END_VAR

VAR_OUTPUT
	OutValue 		: REAL; 			// Output Value
	
END_VAR

VAR 
	TP_Reset 		: TP;				// Maintain reset for 3 seconds
	
	InValue 		: REAL:=0.0 ; 		//  Input Value
 
END_VAR

// RESET //
	TP_Reset(IN := Reset, PT := T#3S);
	
	IF TP_Reset.Q THEN 
		InValue := InitialValue;
		
	END_IF



// RAMP UP //
	IF (Setpoint<(InValue + DeadBand/100*Range)) AND (SetPoint > (InValue-DeadBand/100*Range)) THEN
		// IF values is inside setpoint deadband 
		OutValue :=SetPoint ; 
		
	ELSIF Setpoint > InValue THEN
		// If value is under setpoint value
		OutValue := MIN(InValue + Slope/100*Range * CycleTime/1000, SetPoint) ; 
		
	ELSE
		// If value is above setpoint value
		OutValue := MAX(InValue - Slope/100*Range * CycleTime/1000, SetPoint) ; 	
		
	END_IF

InValue :=OutValue ;

END_FUNCTION_BLOCK

// ---- 00_FunctionsBlocks/Common/DataProcessing/MergeWord/FB_ISKRA_T5.TcPOU
FUNCTION_BLOCK FB_ISKRA_T5
// FB Utilisée uniquement pour motherfucking ISKRA de mes couilles.... 
// 
VAR_INPUT

	WORD_WEAK		: WORD;				// Strong Word. Word to consider if size equals 1.
	WORD_STRONG		: WORD;
END_VAR
VAR_OUTPUT
	VAR_OUT			: REAL;
END_VAR
VAR
	FullWord		: DWORD;
	ValExp			: SINT;
	ValCorps		: UDINT;
END_VAR


FullWord := SHL(WORD_TO_DWORD(WORD_STRONG), 16) OR WORD_Weak;

ValExp := BYTE_TO_SINT(DWORD_TO_BYTE(SHR(FullWord, 24)));
ValCorps := DWORD_TO_UDINT(SHR(SHL(FullWord, 8),8));

VAR_OUT :=  ValCorps*EXPT(10, ValExp);

END_FUNCTION_BLOCK

// ---- 00_FunctionsBlocks/Common/DataProcessing/MergeWord/FB_ISKRA_T6.TcPOU
FUNCTION_BLOCK FB_ISKRA_T6
// FB Utilisée uniquement pour motherfucking ISKRA de mes couilles.... 
// 
VAR_INPUT

	WORD_WEAK		: WORD;				// Strong Word. Word to consider if size equals 1.
	WORD_STRONG		: WORD;
END_VAR
VAR_OUTPUT
	VAR_OUT			: REAL;
END_VAR
VAR
	
	Filtre			: DWORD := 2#11111111000000000000000000000000;
	FullWord		: DWORD;
	ValExp			: SINT;
	ValCorps		: DINT;
	
END_VAR


FullWord := SHL(WORD_TO_DWORD(WORD_STRONG), 16) OR WORD_Weak;

ValExp := BYTE_TO_SINT(DWORD_TO_BYTE(SHR(FullWord, 24)));

ValCorps := -DWORD_TO_DINT(NOT (FullWord OR Filtre) + 1);


VAR_OUT :=  ValCorps*EXPT(10, ValExp);

END_FUNCTION_BLOCK

// ---- 00_FunctionsBlocks/Common/DataProcessing/MergeWord/FB_MergeWordsToUlint.TcPOU
FUNCTION_BLOCK FB_MergeWordsToUlint
////////////////// 
// Merge two words or one word into a DINT or UDINT with big endian coding. And finally Output a Real. 
//////////////////	

VAR_IN_OUT
	VAR_OUT 		: ULINT ; 	
	
END_VAR

VAR_INPUT
	WORD1 		: WORD; 			// Strong Word. Word to consider if size equals 1.
	WORD2 		: WORD 	:= 0; 		// Weak Word. 
	WORD3 		: WORD 	:= 0; 		// Weak Word. 
	WORD4 		: WORD 	:= 0; 		// Weak Word. 
	

END_VAR

VAR
	VAR_AUX 		: ULINT ;			
	
END_VAR



MEMCPY(destAddr := ADR(VAR_OUT)+3*SIZEOF(word1), srcAddr := ADR(WORD1), n := SIZEOF(word1));
MEMCPY(destAddr := ADR(VAR_OUT)+2*SIZEOF(word1), srcAddr := ADR(WORD2), n := SIZEOF(word1));
MEMCPY(destAddr := ADR(VAR_OUT)+1*SIZEOF(word1), srcAddr := ADR(WORD3), n := SIZEOF(word1));
MEMCPY(destAddr := ADR(VAR_OUT)+0*SIZEOF(word1), srcAddr := ADR(WORD4), n := SIZEOF(word1));

END_FUNCTION_BLOCK

// ---- 00_FunctionsBlocks/Common/DataProcessing/SplitWord/FB_SplitDintToWords.TcPOU
FUNCTION_BLOCK FB_SplitDintToWords
////////////////// 
// Convert one REAL into  2 separate WORDS in Big Endian Encoding. 
//////////////////	
VAR_INPUT
	IN		: DINT ;				// Real input
	
END_VAR

VAR_OUTPUT
	OUT		: ARRAY[0..1]OF WORD;	// Word output array
	
END_VAR

OUT[1] := DWORD_TO_WORD(SHR(SHL(DINT_TO_DWORD(IN),16),16)) ; 	// Strong Word
OUT[0] := DWORD_TO_WORD(SHR(DINT_TO_DWORD(IN),16)); 			// Weak Word

END_FUNCTION_BLOCK

// ---- 00_FunctionsBlocks/Common/DataProcessing/SplitWord/FB_SplitWordToByte.TcPOU
FUNCTION_BLOCK FB_SplitWordToByte
////////////////// 
// Convert one REAL into  2 separate WORDS in Big Endian Encoding. 
//////////////////	
VAR_INPUT
	IN		: WORD ;				// Real input
	
END_VAR

VAR_OUTPUT
	STRONG_BYTE		: BYTE;	// Word output array
	WEAK_BYTE		: BYTE;	// Word output array
END_VAR

STRONG_BYTE := WORD_TO_BYTE(IN) ; 				
WEAK_BYTE 	:= WORD_TO_BYTE(SHR(IN,8));

END_FUNCTION_BLOCK

// ---- 00_FunctionsBlocks/Common/DataProcessing/Substring.TcPOU
PROGRAM Substring
// Gives nth occurence of the string encased by delimiter where n = In_Position
//Donne la position de la IN_Position-ième répétition du caractère recherché et renvoie la chaine de caractères suivante
VAR_INPUT
	IN_Delimiter 		: STRING;
	IN_TextToSearch		: T_MaxString;
	IN_Position			: UINT;
END_VAR

VAR
	n					: UINT;	
	Position_Int		: UINT;
	TextToSearch_Int	: T_MaxString;
END_VAR

VAR_OUTPUT
	OUT_NextString			: T_Maxstring;
END_VAR

n:= 0;
TextToSearch_Int := IN_TextToSearch;
Position_Int := INT_TO_UINT( Find(STR1 := TextToSearch_Int, STR2 := IN_Delimiter));


WHILE Position_Int > 0 AND n < IN_Position DO
	OUT_NextString := LEFT(STR := TextToSearch_Int, SIZE := UINT_TO_INT(Position_Int));
	TextToSearch_Int := RIGHT(STR := TextToSearch_Int, SIZE := LEN(STR:= TextToSearch_Int)- LEN(STR := OUT_NextString));
	Position_Int := INT_TO_UINT(FIND(STR1 := TextToSearch_Int, STR2 := IN_Delimiter));
	n := n + 1;
END_WHILE

IF n <> IN_Position THEN
	OUT_NextString := '';
ELSE
	OUT_NextString := left(STR:= OUT_NextString, SIZE := LEN(STR := OUT_NextString) -1);
END_IF

END_PROGRAM

// ---- 00_FunctionsBlocks/Common/HistorizationVisu/FB_OperationIndex.TcPOU
FUNCTION_BLOCK FB_OperationIndex
////////////////// 
// Get Operationnal Indicators . Number of movements. Running hours, Last Move datetime 
//////////////////	
VAR_INPUT
	MesON				: BOOL ; 
	CmdReset			: BOOL ;

END_VAR

VAR_OUTPUT PERSISTENT
	CalRunningTimeHr	: INT ; 	// (Hrs) Running Time  
	CalNbMove			: WORD ;
	CalTimeStart		: STRING 	;	// DateTime at last Move .  ( hour Granularity ) .

END_VAR

VAR PERSISTENT
	CalRunningTime		: TIME ;
	CalRunningTime_Temp	: TIME;		// Previous RunningTime ater last move. 
	CTU 				: CTU ;		// Count the nb of moves 
	
END_VAR 

VAR 
	ElapsedTime 		: TIME ;	//  Elapsed Time since last move 
	CurrentTime 		: TIME ; 	// Current Time 
	TimeStart			: TIME 	;	// TImeHour when the Move starts for the last time
	R_TRIG 				: R_TRIG ; 	// Detect move starts
	F_TRIG 				: F_TRIG ; 	// Detect move stops

END_VAR


// RESET //
	IF CmdReset THEN 
		TimeStart 			:= TIME() ; 
		CalRunningTime 		:= T#0MS ; 
		CalRunningTime_Temp := T#0MS ;
		CTU(CU:=FALSE) ; 
		CTU(RESET:=TRUE); 
	END_IF



// NUMBER OF MOVES //
//	CTU(CU := MesON , RESET:=FALSE , PV:=65535 , CV => CalNbMove ) ; 
	
// RUNNING HOURS //
	R_TRIG(CLK:= MesON ) ; 
	F_TRIG(CLK:= MesON ) ; 
	
	CurrentTime := TIME() ;
	
	IF R_TRIG.Q THEN 
		TimeStart := TIME() ; 
		CalTimeStart := LEFT(sTimeLocal_G, 16);	 // Minutes granularity . 
	END_IF
	
	ElapsedTime 	:= CurrentTime - TimeStart ;	
	IF MesON THEN 
 
		CalRunningTime  := CalRunningTime_Temp +  ElapsedTime ;
		
	ELSE
		CalRunningTime_Temp := CalRunningTime ; 
		
	END_IF

	CalRunningTimeHr	:= DWORD_TO_INT(TIME_TO_DWORD(CalRunningTime)/1000/3600) ;

END_FUNCTION_BLOCK

// ---- 00_FunctionsBlocks/Common/HistorizationVisu/GetTime.TcPOU
PROGRAM GetTime
VAR
	
	// DATETIME //
		FB_GetSystemTime        : GETSYSTEMTIME;
		FB_ToLocal 				: FB_FileTimeToTzSpecificLocalTime;
		fileTime        		: T_FILETIME;
		FileTimeLocal			: T_FILETIME;
	
	//TEST//
		VarTest AT %I* 			: UINT ; 		// Test variable to be linked to ethercat devices before activation to run tests without complete powerplant.
	
END_VAR

	// DateTime 
	FB_GetSystemTime(
		timeLoDW	=> fileTime.dwLowDateTime, 
		timeHiDW	=> fileTime.dwHighDateTime);
		
	FB_ToLocal(
		in			:=fileTime,
		tzInfo 		:= CstTimeZone_G,
		out		 	=> FileTimeLocal);
		
	sTimeGMT_G 		:= SYSTEMTIME_TO_STRING(FILETIME_TO_SYSTEMTIME(fileTime));	// Full Date Time with ms granularity GMT
	sTimeLocal_G	:= SYSTEMTIME_TO_STRING (FILETIME_TO_SYSTEMTIME(FileTimeLocal));

END_PROGRAM

// ---- 00_FunctionsBlocks/Templates/FB_EX_Example.TcPOU
FUNCTION_BLOCK FB_EX_Example
//////////////////
// 
//////////////////
VAR CONSTANT PERSISTENT
	// Characteristics of the object (Same for all instances)
	
END_VAR

VAR_INPUT PERSISTENT
	// Parameters of the Object (instance specific) 
	
END_VAR

VAR_OUTPUT
	//Child objects
	
END_VAR
VAR
	//M_METHOD2 VARIABLES//
	
	
	//M_METHOD2 VARIABLES//
	
	
	//M_METHOD3 VARIABLES//
	
	
	//GET/SET PROPERTY MANAGEMENT//
	
	
END_VAR

END_FUNCTION_BLOCK

// ---- 01_Equipement_Library/Actuators/FB_CB_AuxMVCB.TcPOU
FUNCTION_BLOCK FB_CB_AuxMVCB EXTENDS FB_CB_Base
//////////////////
//  Motorized Circuit Breaker with telecommAND   Requires Open and Close impulsions.
//////////////////

VAR_INPUT PERSISTENT
	// Parameters of the Object (instance/model specific) 
	ParamTP_Impulsion	   : TIME := T#2S;			(* (s)  Config : Tempo for the start or stop command impulsion*)
	ParamFuseNC		       : BOOL;					(* (NA) False: TRUE = Closed , True : TRUE = opened	*)
END_VAR

VAR_OUTPUT
	//Child objects
	
END_VAR

VAR_INPUT
	// I/O Inputs              
	
	IN_MesFuse_IO				: BOOL ;	(* Upstream switch gear                *)
	IN_Opened_IO 				: BOOL ;	(* Upstream melting of fuses contact   *)
	IN_LvSwitch_IO				: BOOL ; 	(* Downstream circuit breaker          *)
	IN_Upstream_Switch_IO		: BOOL ; 	(* LV switch gear PT1 delivery station *)
	IN_Alim_48v_IO				: BOOL ; 	(* 48V switch gear                     *)
	IN_MesEarth_IO				: BOOL; 
	
	
	MesDataExd	: CB_AuxMVCB_Sch;	
END_VAR

VAR
	//M_OPENCLOSE VARIABLES//	
		RsFuse				:RS;
		TPMesFuse			: TP;		
		TPOpened			: TP;		
		TPLVSwitch			: TP;
		TPUpstream			: TP;
		TPAlim48			: TP;
		
		
	//M_ALARMMANAGEMENT VARIABLES//

 
	//M_STATEMANAGER VARIABLES//
	
	// M_EXECUTE VARIABLES //
		
 
END_VAR

METHOD M_AlarmManagement
//////////////////
// Manages Contactor alarms and warnings
/////////////////

VAR 
	// Method local variables (reinitialized at each cycle) 
	FB_AlarmCodeManager			: FB_AlarmCodeManager ; 	
END_VAR
// Check if command and measures are matching after tempo

TON_NotClosedAndNotOpened(IN:=  NOT MesClosed AND NOT MesOpened , PT := ParamTimeOut_Alarm) ; 
TON_ClosedAndOpened(IN:=MesClosed AND MesOpened, PT := ParamTimeOut_Alarm) ; 

RsFuse(Set:= MesDataExd.MesFuseBurned ,Reset1:=GVL_CFG.CmdClearFault_G OR IN_CmdReset);

TPOpened	(IN:= NOT MesDataExd.MesUpstream_Switch	,PT:= ParamTimeOut_Alarm	);
TPMesFuse	(IN:= NOT MesDataExd.MesFuseBurned		,PT:= ParamTimeOut_Alarm	);
TPLVSwitch	(IN:= NOT MesDataExd.MesData.MesOpened	,PT:= ParamTimeOut_Alarm	);
TPUpstream	(IN:= NOT MesDataExd.MesLvSwitch		,PT:= ParamTimeOut_Alarm	);
TPAlim48	(IN:= NOT MesDataExd.MesAlim_48v		,PT:= ParamTimeOut_Alarm	);



 
// ALARM CODE //
	FB_AlarmCodeManager(
		bAlarm1			:= FALSE,										//
		bAlarm2			:= TON_NotClosedAndNotOpened.Q,					// Incoherent state measure (neither open nor closed) 
		bAlarm3 		:= TON_ClosedAndOpened.Q, 						// Incoherent state measure (Open and closed)	
		bAlarm4			:= MesDataExd.MesUpstream_Switch,				// Upstream switch gear  is opened             
		bAlarm5			:= MesDataExd.MesFuseBurned,		    		// Upstream melting of fuses contact  alarm
		bAlarm6			:= MesDataExd.MesData.MesOpened, 				// Downstream circuit breaker Alarm     
		bAlarm7			:= MesDataExd.MesLvSwitch,			            // LV switch gear PT1 delivery station alarm
		bAlarm8			:= MesDataExd.MesAlim_48v,			            // 48V switch gear Alarm                  
		bAlarm9			:= FALSE,                                       //
		bAlarm10		:= FALSE,                                       //
		bAlarm11		:= FALSE,                                       //
		bAlarm12		:= FALSE,                                       //
		bAlarm13		:= FALSE, 										//
		bAlarm14		:= FALSE, 										//
		bAlarm15		:= FALSE , 										// 
		wAlarmCode		=>MesDataExd.MesData.MesAlarmCode);

//WARNING CODE//
		FB_AlarmCodeManager(
		bAlarm1			:= FALSE, 										// 
		bAlarm2			:= FALSE,	 									// 
		bAlarm3 		:= FALSE,										// 
		bAlarm4			:= FALSE, 										// 
		bAlarm5			:= FALSE, 										//
		bAlarm6			:= MesDataExd.MesEarth, 						// The cell is connected to earth (earthing)
		bAlarm7			:= FALSE, 										//
		bAlarm8			:= FALSE,                                       //
		bAlarm9			:= FALSE,                                       //
		bAlarm10		:= FALSE,                                       //
		bAlarm11		:= FALSE,                                       //
		bAlarm12		:= FALSE,                                       //
		bAlarm13		:= FALSE,                                       //
		bAlarm14		:= FALSE,                                       //
		bAlarm15		:= FALSE, 										//
		wAlarmCode 		=>MesDataExd.MesData.MesWarningCode);

// EVENT CODE //
	FB_AlarmCodeManager(
		bAlarm1			:= FALSE, 										// 
		bAlarm2			:= FALSE, 										// 
		bAlarm3			:= MesOpened, 									// Open position
		bAlarm4			:= MesClosed, 									// Closed position
		bAlarm5			:= IN_CmdReset, 								// Reset Command
		bAlarm6			:= TPMesFuse.Q,									// Upstream switch gear  is closed              
		bAlarm7			:= TPOpened.Q,    								// Upstream melting of fuses contact  alarm back to normal 
		bAlarm8			:= TPLVSwitch.Q,								// Downstream circuit breaker Alarm back to normal           
		bAlarm9			:= TPUpstream.Q,       							// LV switch gear PT1 delivery station alarm back to normal
		bAlarm10		:= TPAlim48.Q,        							// 48V switch gear Alarm back to normal                 
		bAlarm11		:= FALSE,										//
		bAlarm12		:= FALSE,                                       //
		bAlarm13		:= FALSE,                                       //
		bAlarm14		:= FALSE, 										//
		bAlarm15		:= FALSE, 										//
		wAlarmCode		=>MesDataExd.MesData.MesEventCode);
		
	// UPDATE STRUCTURE


	IF ParamNC THEN 
		
	MesDataExd.MesFuseBurned 		:= NOT IN_MesFuse_IO			;
	MesDataExd.MesUpstream_Switch	:= NOT IN_Upstream_Switch_IO	;
	MesDataExd.MesData.MesOpened 	:= NOT IN_LvSwitch_IO			;
	MesDataExd.MesLvSwitch			:= NOT IN_Upstream_Switch_IO	;
	MesDataExd.MesAlim_48v			:= NOT IN_Alim_48v_IO			;
	ELSE
	MesDataExd.MesFuseBurned 		:=  IN_MesFuse_IO				;
	MesDataExd.MesUpstream_Switch	:=  IN_Opened_IO 				;
	MesDataExd.MesData.MesOpened 	:=  IN_LvSwitch_IO				;
	MesDataExd.MesLvSwitch			:=  IN_Upstream_Switch_IO		;
	MesDataExd.MesAlim_48v			:=  IN_Alim_48v_IO				;
	END_IF
	
MesDataExd.MesEarth	:= IN_MesEarth_IO ;
END_METHOD

METHOD M_Execute
VAR_INPUT
END_VAR
// PERMANENT CONDITIONS //	
MesDataExd.MesData.MesCP_Open					:= IN_CmdOpen AND NOT IN_CmdReset;
MesDataExd.MesData.MesCP_Close				:= NOT MesDataExd.MesData.MesClosed AND IN_CmdClose AND NOT MesDataExd.MesData.MesAlarmCode.0 AND NOT MesDataExd.MesData.MesCP_Open AND NOT IN_CmdReset ;


SUPER^.M_Execute();
END_METHOD

METHOD M_OpenClose
//////////////////
// Manages Opening and Closing of the contactor
//////////////////

VAR 
	// Method local variables (reinitialized at each cycle) 

	
END_VAR
END_METHOD

METHOD M_StateManager
//////////////////
// Manages Contactor State
/////////////////

VAR 
	// Method local variables (reinitialized at each cycle) 
	
END_VAR
MesState := 0 ; 
IF MesOpened THEN		// If the cell seems opens and closed in the same time, we will consider it as opened. 
	
	MesState.0 := 1 ; 
MesDataExd.MesData.MesClosed := FALSE ; 
MesDataExd.MesData.MesOpened := TRUE ; 
ELSIF MesClosed THEN
	
	MesState.1 := 1 ; 
MesDataExd.MesData.MesClosed := TRUE ; 
MesDataExd.MesData.MesOpened := FALSE ; 
ELSE 
	MesState.0 := 1 ;		// if the cell seems neither opened and neither closed , we will consider it as opened. 
MesDataExd.MesData.MesClosed := FALSE ; 	
MesDataExd.MesData.MesOpened := TRUE ; 
END_IF
END_METHOD

END_FUNCTION_BLOCK

// ---- 01_Equipement_Library/Actuators/FB_CB_Base.TcPOU
FUNCTION_BLOCK FB_CB_Base
//////////////////
// Electrical Switch - Base FB
//////////////////

VAR_INPUT PERSISTENT
	// Parameters of the Object (instance/model specific) 
	ParamTimeOut_Open       		: TIME  := T#1S     ;       (* (ms) Config : Tempo to open before Timeout warning  *)
	ParamTimeOut_Close      		: TIME  := T#1S     ;		(* (ms) Config : Tempo to close before Timeout warning*)
	ParamTimeOut_Alarm   		    : TIME  := T#200MS  ;		(* (ms) Config : Tempo when open and close before raising alarm*)
	ParamNC							: BOOL  := FALSE    ;		(* (NA) False: TRUE = Closed, True : TRUE = opened*)
	ParamNbFdbck			    	: BYTE  := 1        ;		(* (NA) Number of feedback position (1: 1 wire, 2 : 2 wire)*)
	ParamClosedInput_Connected		: BOOL  := TRUE     ; 		(* (NA) True : closed input is connected*)
	                                                    	
END_VAR

VAR_OUTPUT
	//Child objects
	
END_VAR

VAR_INPUT
	// I/O Inputs 
		IN_MesOpened_IO					: BOOL  ; 				// (NA) [P,H,B] Opened Position IO	         
		IN_MesClosed_IO 				: BOOL := TRUE ; 		// (NA) [P,H,B] Closed Position IO           
	
		IN_CmdOpen 						: BOOL ; 				// (NA) External Open Command 
		IN_CmdClose						: BOOL ; 				// (NA) External Close Command 
		
	{attribute 'OPC.UA.DA' := '1'}   
		IN_CmdReset					: BOOL ;				// (NA) External Reset Command              // Check: what does the L respresent ? 
END_VAR

VAR
	//M_OPENCLOSE VARIABLES//
		MesOpened					     : BOOL ;                                                                     
		MesClosed					     : BOOL ;                                                                     
		
	//M_ALARMMANAGEMENT VARIABLES//
		FB_CheckCommand				     : FB_CheckCommand ; 	//(NA) Check if start command successful 
		FB_CheckCommand2			     : FB_CheckCommand ;	//(NA) Check if stop command successful  
		TON_ClosedAndOpened			     : TON ;              	
		TON_NotClosedAndNotOpened	     : TON ;              	
                                             	
		
		
	//M_STATEMANAGER VARIABLES//
		MesState					     : BYTE ; 				// (NA) Cal [P,H,B] Bit 0: Open , Bit 1: Closed        
	///MesDataExd				     : CB ; 

	// M_EXECUTE VARIABLES 	//                                   
		MesCP_Open		: BOOL ;   	(* Cal(NA) Permanent Conditions*)
		MesCP_Close		: BOOL ; 	(* Cal(NA) Permanent Conditions*) 

	//M_EMULATOR
	
		CmdExternalClose_Emul		: BOOL;
		CmdExternalOpen_Emul		: BOOL;
		
		RS_Emulate					: RS;
		
		TON_OutputWait_Open			: TON;
		TON_OutputWait_Close		: TON;
		
		R_TRIGOpen					: R_TRIG;
		R_TRIGClose					: R_TRIG;
			
END_VAR

METHOD M_AlarmManagement
//////////////////
// Manages Contactor alarms and warnings
/////////////////

VAR 
	// Method local variables (reinitialized at each cycle) 

	
END_VAR
END_METHOD

METHOD M_Emulator
VAR_INPUT
END_VAR
END_METHOD

METHOD M_Execute
VAR_INPUT
END_VAR
// If One wire feedback , Open Position is the inverse of Close Position. 
	IF  ParamNbFdbck=1 AND ParamClosedInput_Connected THEN
		IN_MesOpened_IO := NOT IN_MesClosed_IO ;
	ELSIF ParamNbFdbck = 1 AND NOT ParamClosedInput_Connected THEN
		IN_MesClosed_IO := NOT IN_MesOpened_IO;
	END_IF
	
	IF ParamNC THEN 
		MesOpened := NOT IN_MesOpened_IO ; 
		MesClosed := NOT IN_MesClosed_IO ; 
	ELSE
		MesOpened := IN_MesOpened_IO ; 
		MesClosed := IN_MesClosed_IO ; 		
	END_IF
	
	
//Methods call	
	M_OpenClose(); 
	M_StateManager() ;
	M_AlarmManagement(); 
	M_Emulator();
END_METHOD

METHOD M_OpenClose
//////////////////
// Manages Opening of the contactor
//////////////////

VAR 
	// Method local variables (reinitialized at each cycle) 
	
END_VAR
END_METHOD

METHOD M_StateManager
//////////////////
// Manages Contactor State
/////////////////

VAR 
	// Method local variables (reinitialized at each cycle) 
	
END_VAR
END_METHOD

END_FUNCTION_BLOCK

// ---- 01_Equipement_Library/Actuators/FB_CB_GridMVCB.TcPOU
FUNCTION_BLOCK FB_CB_GridMVCB EXTENDS FB_CB_Base
//////////////////
//  Motorized Circuit Breaker with telecommAND   Requires Open and Close impulsions.
//////////////////

VAR_INPUT PERSISTENT
	// Parameters of the Object (instance/model specific) 
	
END_VAR

VAR_INPUT
	// I/O Inputs              	
	MesDataExd			: CB_Standard ; 	
END_VAR

VAR
	//M_OPENCLOSE VARIABLES//

	
	//M_ALARMMANAGEMENT VARIABLES//
		
	//M_STATEMANAGER VARIABLES//

	// M_EXECUTE VARIABLES //
		
	

		
END_VAR

METHOD M_AlarmManagement
//////////////////
// Manages Contactor alarms and warnings
/////////////////

VAR 
	// Method local variables (reinitialized at each cycle) 
	FB_AlarmCodeManager			: FB_AlarmCodeManager ; 

	
END_VAR
VAR_INPUT
	
END_VAR
// Check if command and measures are matching after tempo
TON_NotClosedAndNotOpened(IN:=  NOT MesClosed AND NOT MesOpened , PT := ParamTimeOut_Alarm) ; 
TON_ClosedAndOpened(IN:= MesClosed AND MesOpened, PT := ParamTimeOut_Alarm) ; 
//RS_AlarmStopReclose(Set := MesTransfo_Fault, RESET1 := BlockWriteTemp[1] OR IN_CmdReset_L);

// ALARM CODE //
	FB_AlarmCodeManager(
		bAlarm1			:= FALSE, 									// 
		bAlarm2			:= TON_NotClosedAndNotOpened.Q,				// Incoherent State measure (Not Opened and not Closed )
		bAlarm3 		:= TON_ClosedAndOpened.Q,	 				// Incoherent State measure (Opened and Closed )	
		bAlarm4			:= FALSE, 									// 
		bAlarm5			:= FALSE, 									//
		bAlarm6			:= FALSE,                                   //
		bAlarm7			:= FALSE,                                   //
		bAlarm8			:= FALSE,                                   //
		bAlarm9			:= FALSE,                                   //
		bAlarm10		:= FALSE,                                   //
		bAlarm11		:= FALSE,                                   //
		bAlarm12		:= FALSE,                                   //
		bAlarm13		:= FALSE, 									//
		bAlarm14		:= FALSE, 									//
		bAlarm15		:= FALSE, 									// 
		wAlarmCode		=>MesDataExd.MesData.MesAlarmCode);

//WARNING CODE //
		FB_AlarmCodeManager(
		bAlarm1			:= FALSE, 									//
		bAlarm2			:= FALSE,	 		                        //
		bAlarm3 		:= FALSE,									//		
		bAlarm4			:= FALSE, 									//
		bAlarm5			:= FALSE,                                   //
		bAlarm6			:= FALSE,                                   //
		bAlarm7			:= FALSE,                                   //
		bAlarm8			:= FALSE,                                   //
		bAlarm9			:= FALSE,                                   //
		bAlarm10		:= FALSE,                                   //
		bAlarm11		:= FALSE,                                   //
		bAlarm12		:= FALSE,                                   //
		bAlarm13		:= FALSE,                                   //
		bAlarm14		:= FALSE,                                   //
		bAlarm15		:= FALSE,                                   //
		wAlarmCode 		=>MesDataExd.MesData.MesWarningCode);

// EVENT CODE //
	FB_AlarmCodeManager(
		bAlarm1			:= FALSE, 									// 
		bAlarm2			:= FALSE, 									// 
		bAlarm3			:= MesOpened, 								// Opened Position
		bAlarm4			:= MesClosed, 								// Closed Position
		bAlarm5			:= IN_CmdReset,                           // Reset Command
		bAlarm6			:= FALSE,                                   //
		bAlarm7			:= FALSE,                                   //
		bAlarm8			:= FALSE,                                   //
		bAlarm9			:= FALSE,                                   //
		bAlarm10		:= FALSE,                                   //
		bAlarm11		:= FALSE,                                   //
		bAlarm12		:= FALSE,                                   //
		bAlarm13		:= FALSE,                                   //
		bAlarm14		:= FALSE,                                   //
		bAlarm15		:= FALSE,                                   //
		wAlarmCode		=>MesDataExd.MesData.MesEventCode);
END_METHOD

METHOD M_Execute
VAR_INPUT
END_VAR
// PERMANENT CONDITIONS //	
MesDataExd.MesData.MesCP_Open					:= IN_CmdOpen AND NOT IN_CmdReset;
MesDataExd.MesData.MesCP_Close				:= NOT MesDataExd.MesData.MesClosed AND IN_CmdClose AND NOT MesDataExd.MesData.MesAlarmCode.0 AND NOT MesDataExd.MesData.MesCP_Open AND NOT IN_CmdReset ;



SUPER^.M_Execute();
END_METHOD

METHOD M_StateManager
//////////////////
// Manages Contactor State
/////////////////

VAR 
	// Method local variables (reinitialized at each cycle) 
	
END_VAR
MesState := 0 ; 
IF MesOpened THEN		// If the cell seems opens and closed in the same time, we will consider it as opened. 
	
	MesState.0 := 1 ; 
MesDataExd.MesData.MesClosed := FALSE ; 
MesDataExd.MesData.MesOpened := TRUE ; 
ELSIF MesClosed THEN
	
	MesState.1 := 1 ; 
MesDataExd.MesData.MesClosed := TRUE ; 
MesDataExd.MesData.MesOpened := FALSE ; 
ELSE 
	MesState.0 := 1 ;		// if the cell seems neither opened and neither closed , we will consider it as opened. 
MesDataExd.MesData.MesClosed := FALSE ; 	
MesDataExd.MesData.MesOpened := TRUE ; 
END_IF
END_METHOD

END_FUNCTION_BLOCK

// ---- 01_Equipement_Library/Actuators/FB_CB_MainHVCB.TcPOU
FUNCTION_BLOCK FB_CB_MainHVCB EXTENDS FB_CB_Base
//////////////////
//  Motorized Circuit Breaker with telecommAND  Requires Open and Close impulsions.
//////////////////

VAR_INPUT PERSISTENT
	// Parameters of the Object (instance/model specific) 
	ParamTP_Impulsion		    : TIME 		:= T#2S ;	(* (s) Config : Tempo for the start or stop command impulsion											*)
	ParamComutNc			    : BOOL ;                (**)
	ParamSectLigne			    : BYTE      :=1 ;		(* (NA) Monitoring du sectionneur de ligne de la MainMVCB.0 = TRUE := Monitoré .1 = TRUE Close is connected, .2 = ParamNC*)

END_VAR

VAR_OUTPUT
	//Child objects
	
END_VAR

VAR_INPUT
	A1_Sect				       : FB_CB_MVSwitch;

// I/O Inputs              
	IN_MesAlarmPwr_IO		           : BOOL ;	              // (NA)[P,H,B] Remote control Power supply Error .  IO  	
	IN_MesTripped_IO		  		   : BOOL ; 	          // Tripped position of the CB Must Ack To switch in again
	IN_MesComut_IO			   	   : BOOL := TRUE ; 	  // True if cell is in local position . 
	IN_MesEarth_IO 			       : BOOL ; 	
	
	MesDataExd	        :  CB_MainHVCB_Sch ; 
	
END_VAR

VAR
	//M_OPENCLOSE VARIABLES//	
	TP_Open	 			: TP ;				// (NA) Temporisation for Open pulse Command
	TP_Close 				: TP ;				// (NA) Temporisation for Close pulse Command	

	//M_ALARMMANAGEMENT VARIABLES//

	
//M_STATEMANAGER VARIABLES//
	
END_VAR

METHOD M_AlarmManagement
//////////////////
// Manages Contactor alarms and warnings
/////////////////

VAR 
	// Method local variables (reinitialized at each cycle) 
	FB_AlarmCodeManager			: FB_AlarmCodeManager ; 
	
	CmdOpenCloseIO: BOOL; //Check IN/OUT_CMDOpenClose
END_VAR


TON_NotClosedAndNotOpened(IN:=  NOT MesClosed AND NOT MesOpened , PT := ParamTimeOut_Alarm) ; 
TON_ClosedAndOpened(IN:=MesClosed AND MesOpened, PT := ParamTimeOut_Alarm) ; 


// ALARM CODE //
	FB_AlarmCodeManager(
		bAlarm1			:= MesDataExd.MesTripped,					// Cb is tripped
		bAlarm2			:= TON_NotClosedAndNotOpened.Q,				// Incoherent State measure (Not Opened and not Closed )
		bAlarm3 		:= TON_ClosedAndOpened.Q   , 				// Incoherent State measure (Opened and Closed )	
		bAlarm4			:= FALSE, 				// 
		bAlarm5			:= FALSE  , 			// 
		bAlarm6			:= FALSE,                                   //
		bAlarm7			:= FALSE,                                   //
		bAlarm8			:= FALSE,                                   //
		bAlarm9			:= FALSE,                                   //
		bAlarm10		:= FALSE,                                   //
		bAlarm11		:= FALSE,                                   //
		bAlarm12		:= FALSE,                                   //
		bAlarm13		:= FALSE,                                   //
		bAlarm14		:= FALSE,                                   //
		bAlarm15		:= FALSE , 									//
		wAlarmCode		=>MesDataExd.MesData.MesAlarmCode);

//WARNING CODE//
		FB_AlarmCodeManager(
		bAlarm1			:= FALSE,//
		bAlarm2			:= FALSE,//
		bAlarm3 		:= FALSE,										// 
		bAlarm4			:= MesDataExd.MesAlarmPwr, 						// Power Supply Fault
		bAlarm5			:= MesDataExd.MesComutLocal, 					// Commutator in local mode 
		bAlarm6			:= MesDataExd.MesEarth, 							// The cell is connected to earth (earthing)
		bAlarm7			:= SEL( ParamSectLigne.0 ,FALSE ,  NOT A1_Sect.MesDataExd.MesData.MesClosed),				// Line connector is opened (sectionneur)
		bAlarm8			:= FALSE, 										//
		bAlarm9			:= FALSE,                                       //
		bAlarm10		:= FALSE,                                       //
		bAlarm11		:= FALSE,                                       //
		bAlarm12		:= FALSE,                                       //
		bAlarm13		:= FALSE,                                       //
		bAlarm14		:= FALSE,                                       //
		bAlarm15		:= FALSE, 										//
		wAlarmCode 		=>MesDataExd.MesData.MesWarningCode);

// EVENT CODE //
	FB_AlarmCodeManager(
		bAlarm1			:= FALSE, 			// 
		bAlarm2			:= FALSE, 		    // 
		bAlarm3			:= MesOpened, 				// Opened Position
		bAlarm4			:= MesClosed, 				// Closed Position
		bAlarm5			:= IN_CmdReset, 			// Reset command
		bAlarm6			:= FALSE, 					//
		bAlarm7			:= FALSE,                   //
		bAlarm8			:= FALSE,                   //
		bAlarm9			:= FALSE,                   //
		bAlarm10		:= FALSE,                   //
		bAlarm11		:= FALSE,                   //
		bAlarm12		:= FALSE,                   //
		bAlarm13		:= FALSE, 					//
		bAlarm14		:= FALSE,                   //
		bAlarm15		:= FALSE,                   //
		wAlarmCode		=>MesDataExd.MesData.MesEventCode);   
		                                            
	//                                              
	                                                
	// UPDATE STRUCTURE

	IF ParamComutNc THEN
	MesDataExd.MesComutLocal	:= NOT IN_MesComut_IO ; 
	ELSE
	MesDataExd.MesComutLocal	:= IN_MesComut_IO ; 
	END_IF
	
MesDataExd.MesAlarmPwr		    := IN_MesAlarmPwr_IO ; 
MesDataExd.MesTripped			:= IN_MesTripped_IO ; 
MesDataExd.MesEarth			    := IN_MesEarth_IO ; 
MesDataExd.MesOpened_Sect	        := SEL(ParamSectLigne.0 , FALSE  , NOT A1_Sect.MesDataExd.MesData.MesClosed ) ;
END_METHOD

METHOD M_Execute
VAR_INPUT
END_VAR

VAR

END_VAR
//MainMVCB avec etat de sectionneur de ligne
IF ParamSectLigne.0 THEN 
	A1_Sect.ParamNbFdbck := 1;
	A1_Sect.ParamNC := ParamSectLigne.2;
	A1_Sect.ParamClosedInput_Connected := ParamSectLigne.1 ; 
	A1_Sect.M_Execute();
END_IF

// PERMANENT CONDITIONS //	
MesDataExd.MesData.MesCP_Open					:= IN_CmdOpen AND NOT IN_CmdReset;
MesDataExd.MesData.MesCP_Close				:= NOT MesDataExd.MesData.MesClosed AND IN_CmdClose AND NOT MesDataExd.MesData.MesAlarmCode.0 AND NOT MesDataExd.MesData.MesCP_Open AND NOT IN_CmdReset ;


SUPER^.M_Execute();
END_METHOD

METHOD M_StateManager
//////////////////
// Manages Contactor State
/////////////////

VAR 
	// Method local variables (reinitialized at each cycle) 
	
END_VAR
MesState := 0 ; 
IF MesOpened THEN		// If the cell seems opens and closed in the same time, we will consider it as opened. 
	
	MesState.0 := 1 ; 
MesDataExd.MesData.MesClosed := FALSE ; 
MesDataExd.MesData.MesOpened := TRUE ; 
ELSIF MesClosed THEN
	
	MesState.1 := 1 ; 
MesDataExd.MesData.MesClosed := TRUE ; 
MesDataExd.MesData.MesOpened := FALSE ; 
ELSE 
	MesState.0 := 1 ;		// if the cell seems neither opened and neither closed , we will consider it as opened. 
MesDataExd.MesData.MesClosed := FALSE ; 	
MesDataExd.MesData.MesOpened := TRUE ; 
END_IF
END_METHOD

END_FUNCTION_BLOCK

// ---- 01_Equipement_Library/Actuators/FB_CB_MVSwitch.TcPOU
FUNCTION_BLOCK FB_CB_MVSwitch EXTENDS FB_CB_Base
//////////////////
//  Motorized Circuit Breaker with telecommAND   Requires Open and Close impulsions.
//////////////////

VAR_INPUT PERSISTENT
	// Parameters of the Object (instance/model specific) 
	
END_VAR

VAR_INPUT
	// I/O Inputs              	
		MesDataExd	       			 :  CB_Standard ; 
END_VAR

VAR
	//M_OPENCLOSE VARIABLES//

	
	//M_ALARMMANAGEMENT VARIABLES//
		
	//M_STATEMANAGER VARIABLES//

	// M_EXECUTE VARIABLES //
		
	// EMULATOR //

		
END_VAR

METHOD M_AlarmManagement
//////////////////
// Manages Contactor alarms and warnings
/////////////////

VAR 
	// Method local variables (reinitialized at each cycle) 
	FB_AlarmCodeManager			: FB_AlarmCodeManager ; 

	
END_VAR
VAR_INPUT
	
END_VAR
// Check if command and measures are matching after tempo
TON_NotClosedAndNotOpened(IN:=  NOT MesClosed AND NOT MesOpened , PT := ParamTimeOut_Alarm) ; 
TON_ClosedAndOpened(IN:= MesClosed AND MesOpened, PT := ParamTimeOut_Alarm) ; 
//RS_AlarmStopReclose(Set := MesTransfo_Fault, RESET1 := BlockWriteTemp[1] OR IN_CmdReset_L);

// ALARM CODE //
	FB_AlarmCodeManager(
		bAlarm1			:= FALSE, 									// 
		bAlarm2			:= TON_NotClosedAndNotOpened.Q,				// Incoherent State measure (Not Opened and not Closed )
		bAlarm3 		:= TON_ClosedAndOpened.Q  , 				// Incoherent State measure (Opened and Closed )	
		bAlarm4			:= FALSE, 									// 
		bAlarm5			:= FALSE, 									//
		bAlarm6			:= FALSE,                                   //
		bAlarm7			:= FALSE,                                   //
		bAlarm8			:= FALSE,                                   //
		bAlarm9			:= FALSE,                                   //
		bAlarm10		:= FALSE,                                   //
		bAlarm11		:= FALSE,                                   //
		bAlarm12		:= FALSE,                                   //
		bAlarm13		:= FALSE, 									//
		bAlarm14		:= FALSE, 									//
		bAlarm15		:= FALSE , 									// 
		wAlarmCode		=>MesDataExd.MesData.MesAlarmCode);

//WARNING CODE//
		FB_AlarmCodeManager(
		bAlarm1			:= FALSE , 									//
		bAlarm2			:= FALSE  , 		                        //
		bAlarm3 		:= FALSE,									//		
		bAlarm4			:= FALSE, 									//
		bAlarm5			:= FALSE,                                   //
		bAlarm6			:= FALSE,                                   //
		bAlarm7			:= FALSE,                                   //
		bAlarm8			:= FALSE,                                   //
		bAlarm9			:= FALSE,                                   //
		bAlarm10		:= FALSE,                                   //
		bAlarm11		:= FALSE,                                   //
		bAlarm12		:= FALSE,                                   //
		bAlarm13		:= FALSE,                                   //
		bAlarm14		:= FALSE,                                   //
		bAlarm15		:= FALSE,                                   //
		wAlarmCode 		=>MesDataExd.MesData.MesWarningCode);

// EVENT CODE //
	FB_AlarmCodeManager(
		bAlarm1			:= FALSE, 									// 
		bAlarm2			:= FALSE, 									// 
		bAlarm3			:= MesOpened, 								// Opened Position
		bAlarm4			:= MesClosed, 								// Closed Position
		bAlarm5			:= IN_CmdReset,                           // Reset Command
		bAlarm6			:= FALSE,                                   //
		bAlarm7			:= FALSE,                                   //
		bAlarm8			:= FALSE,                                   //
		bAlarm9			:= FALSE,                                   //
		bAlarm10		:= FALSE,                                   //
		bAlarm11		:= FALSE,                                   //
		bAlarm12		:= FALSE,                                   //
		bAlarm13		:= FALSE,                                   //
		bAlarm14		:= FALSE,                                   //
		bAlarm15		:= FALSE,                                   //
		wAlarmCode		=>MesDataExd.MesData.MesEventCode);
END_METHOD

METHOD M_Execute
VAR_INPUT
END_VAR
// PERMANENT CONDITIONS //	
MesDataExd.MesData.MesCP_Open					:= IN_CmdOpen AND NOT IN_CmdReset;
MesDataExd.MesData.MesCP_Close				:= NOT MesDataExd.MesData.MesClosed AND IN_CmdClose AND NOT MesDataExd.MesData.MesAlarmCode.0 AND NOT MesDataExd.MesData.MesCP_Open AND NOT IN_CmdReset ;


SUPER^.M_Execute();
END_METHOD

METHOD M_StateManager
//////////////////
// Manages Contactor State
/////////////////

VAR 
	// Method local variables (reinitialized at each cycle) 
	
END_VAR
MesState := 0 ; 
IF MesOpened THEN		// If the cell seems opens and closed in the same time, we will consider it as opened. 
	
	MesState.0 := 1 ; 
MesDataExd.MesData.MesClosed := FALSE ; 
MesDataExd.MesData.MesOpened := TRUE ; 
ELSIF MesClosed THEN
	
	MesState.1 := 1 ; 
MesDataExd.MesData.MesClosed := TRUE ; 
MesDataExd.MesData.MesOpened := FALSE ; 
ELSE 
	MesState.0 := 1 ;		// if the cell seems neither opened and neither closed , we will consider it as opened. 
MesDataExd.MesData.MesClosed := FALSE ; 	
MesDataExd.MesData.MesOpened := TRUE ; 
END_IF
END_METHOD

END_FUNCTION_BLOCK

// ---- 01_Equipement_Library/Actuators/FB_CB_MainMVCB.TcPOU
FUNCTION_BLOCK FB_CB_MainMVCB EXTENDS FB_CB_Base
//////////////////
//  Motorized Circuit Breaker with telecommAND  Requires Open and Close impulsions.
//////////////////

VAR_INPUT PERSISTENT
	// Parameters of the Object (instance/model specific) 
	ParamTP_Impulsion		    : TIME 		:= T#2S;	(* (s) Config : Tempo for the start or stop command impulsion*)
	ParamComutNc			    : BOOL;					(* (NA) Local selector in normally closed. NC >> True = Selector in local *)
	ParamSectLigne			    : BYTE      :=1;		(* (NA) Monitoring du sectionneur de ligne de la MainMVCB . 0 = TRUE := Monitoré . 1 = TRUE Close is connected*)
	ParamUvCoil					: BOOL;					(* (NA) if the open and close order are linked to a undervoltage coil (Bobine à manque, Bobine Mn), this should be True*)
	ParamAlarmPwr_NC			: BOOL;
END_VAR

VAR_OUTPUT
	//Child objects
	OUT_CmdOpen_IO	           : BOOL ; 	          // (NA) Physical I/O Open Command IO
	OUT_CmdClose_IO			   : BOOL ; 	          // (NA) Physical I/O Close Command IO
	OUT_CmdMaintainClose_IO		: BOOL;					// (NA) Physical I/O close for the UV coil.
END_VAR

VAR_INPUT
	A1_Sect				        : FB_CB_MVSwitch;

// I/O Inputs              
	IN_MesAlarmPwr_IO		    : BOOL ;	          // (NA)[P,H,B] Remote control Power supply Error  IO  	
	IN_MesTripped_IO		  	: BOOL ; 	          // (NA) Tripped position of the CB Must Ack To switch in again
	IN_MesComutLocal_IO			: BOOL := TRUE ; 	  // (NA) True if cell is in local position  
	IN_MesEarth_IO 			    : BOOL ;
	IN_MesRSE_IO				: BOOL ;  	

	IN_MesSwitchG_IO			: BOOL ; 	  		    
	IN_MesTest_Serv_IO 			: BOOL ;		
	IN_MesOpened_Sect_IO 		: BOOL ;		
	IN_MesDefaulr_48VCC_IO		: BOOL ; 	
	
	
	
	
//M_Emulator
	IN_GTE_Default_Emul			: BOOL;
	
	TON_GTE_Default_Emul		: TON;
	
	MesDataExd			        :  CB_MainMVCB_Sch ; 
		
END_VAR

VAR
	//M_OPENCLOSE VARIABLES//	
		ParamTP_Open	 			: TP ;				(* (NA) Temporisation for Open pulse Command*)
		ParamTP_Close 				: TP ;				(* (NA) Temporisation for Close pulse Command	*)
		RS_MaintainClose			: RS ;				(* (NA) RS to manage UV Coil*)

		TP_Opened					: TP ;
		TP_ComutLocal				: TP ;
		TP_SwitchG		            : TP ;
		TP_Test_Serv 	            : TP ;
		TP_Opened_Sect 	            : TP ;
		TP_Defaulr_48VCC            : TP ;
		
		
		
		
	//M_ALARMMANAGEMENT VARIABLES//
	
//M_STATEMANAGER VARIABLES//
	
END_VAR

METHOD M_AlarmManagement
//////////////////
// Manages Contactor alarms and warnings
/////////////////

VAR 
	// Method local variables (reinitialized at each cycle) 
	FB_AlarmCodeManager			: FB_AlarmCodeManager ; 
	
	CmdOpenCloseIO				: BOOL; 				//Check IN/OUT_CMDOpenClose
	bSectLigne					: BOOL;
END_VAR
// Check if command and measures are matching after tempo
FB_CheckCommand	(T:= ParamTimeOut_Close, bCmd:=OUT_CmdClose_IO , bMes := MesDataExd.MesData.MesClosed , bImpulsion := FALSE , bReset := CmdClearFault_G OR OUT_CmdClose_IO) ; 
FB_CheckCommand2(T:= ParamTimeOut_Open , bCmd:= OUT_CmdOpen_IO , bMes :=NOT MesDataExd.MesData.MesClosed , bImpulsion := FALSE , bReset := CmdClearFault_G OR OUT_CmdOpen_IO) ; 

TON_NotClosedAndNotOpened(IN:=  NOT MesClosed AND NOT MesOpened , PT := ParamTimeOut_Alarm) ; 
TON_ClosedAndOpened(IN:=MesClosed AND MesOpened, PT := ParamTimeOut_Alarm) ; 



TP_Opened			(IN:= NOT MesDataExd.MesData.MesOpened 		,PT:= ParamTimeOut_Alarm	);	
TP_ComutLocal		(IN:= NOT MesDataExd.MesComutLocal	    	,PT:= ParamTimeOut_Alarm	);	
TP_SwitchG		    (IN:= NOT MesDataExd.MesSwitchG		      	,PT:= ParamTimeOut_Alarm	);
TP_Test_Serv 	    (IN:= NOT MesDataExd.MesTest_Serv 	    	,PT:= ParamTimeOut_Alarm	);
TP_Opened_Sect 	    (IN:= NOT MesDataExd.MesOpened_Sect 	  	,PT:= ParamTimeOut_Alarm	);
TP_Defaulr_48VCC 	(IN:= NOT MesDataExd.MesDefaulr_48VCC	 	,PT:= ParamTimeOut_Alarm	);

// ALARM CODE //

// Attention une alarm doit être mise en commentaire de la manière suivante (* *), l'utilisation du // pose pb sur Bazefield 

	FB_AlarmCodeManager(
		bAlarm1			:= MesDataExd.MesTripped,						// Cb is tripped
		bAlarm2			:= TON_NotClosedAndNotOpened.Q,					// Incoherent State measure (Not Opened and not Closed)
		bAlarm3 		:= TON_ClosedAndOpened.Q,	 					// Incoherent State measure (Opened and Closed)	
		bAlarm4			:= FB_CheckCommAND.bWarning, 					// Close command failed
		bAlarm5			:= FB_CheckCommand2.bWarning,	 				// Open Command failed
		bAlarm6			:= MesDataExd.MesData.MesOpened ,               // Circuit breaker is opened      
		bAlarm7			:= MesDataExd.MesComutLocal	    ,               // Local/remote operation
		bAlarm8			:= MesDataExd.MesSwitchG		,               // Plant switch gear is Opened  
		bAlarm9			:= MesDataExd.MesTest_Serv 	    ,               // test/service          
		bAlarm10		:= MesDataExd.MesOpened_Sect 	,               // Utility switch gear is opened
		bAlarm11		:= MesDataExd.MesDefaulr_48VCC	,               // 48Vcc default         
		bAlarm12		:= FALSE,                                   	//
		bAlarm13		:= FALSE,                                   	//
		bAlarm14		:= FALSE,                                   	//
		bAlarm15		:= FALSE , 										//
		wAlarmCode		=>MesDataExd.MesData.MesAlarmCode);

	//bSectLigne := SEL(ParamSectLigne.0 ,FALSE , NOT A1_Sect.MesDataExd.MesData.MesClosed);
//WARNING CODE//
		FB_AlarmCodeManager(
		bAlarm1			:= FALSE,										//
		bAlarm2			:= FALSE,										//
		bAlarm3 		:= FALSE,										// 
		bAlarm4			:= MesDataExd.MesAlarmPwr, 						// Power Supply Fault
		bAlarm5			:= MesDataExd.MesComutLocal, 					// Commutator in local mode 
		bAlarm6			:= MesDataExd.MesEarth, 						// The cell is connected to earth (earthing)
		bAlarm7			:= bSectLigne,									// Line connector is opened (sectionneur)
		bAlarm8			:= FALSE, 										//
		bAlarm9			:= FALSE,                                       //
		bAlarm10		:= FALSE,                                       //
		bAlarm11		:= FALSE,                                       //
		bAlarm12		:= FALSE,                                       //
		bAlarm13		:= FALSE,                                       //
		bAlarm14		:= FALSE,                                       //
		bAlarm15		:= FALSE, 										//
		wAlarmCode 		=>MesDataExd.MesData.MesWarningCode);

// EVENT CODE //
	FB_AlarmCodeManager(
		bAlarm1			:= OUT_CmdOpen_IO, 								// Open Command
		bAlarm2			:= OUT_CmdClose_IO, 							// Close Command
		bAlarm3			:= MesOpened, 									// Opened Position
		bAlarm4			:= MesClosed, 									// Closed Position
		bAlarm5			:= IN_CmdReset, 								// Reset command
		bAlarm6			:= MesDataExd.MesComutLocal	    ,               // Local mode is activated
		bAlarm7			:= TP_ComutLocal.Q		    ,           		// Remote operation is activated
		bAlarm8			:= MesDataExd.MesTest_Serv 	    ,               // Test mode is activated  
		bAlarm9			:= TP_Test_Serv.Q 	    ,           			// Service  mode is activated
		bAlarm10		:= TP_Opened.Q,                   				// Circuit breaker is closed
		bAlarm11		:= TP_SwitchG.Q,                   				// Plant switch gear is closed
		bAlarm12		:= TP_Opened_Sect.Q,                   			// Utility switch gear is closed
		bAlarm13		:= TP_Defaulr_48VCC.Q, 							// 48Vcc default alarm back to normal
		bAlarm14		:= FALSE,                   					//
		bAlarm15		:= FALSE,                   					//
		wAlarmCode		=>MesDataExd.MesData.MesEventCode);                                               
	                                                
	// UPDATE STRUCTURE
	
	IF ParamNc THEN
	MesDataExd.MesData.MesOpened	:= NOT IN_MesOpened_IO		    ; 
	MesDataExd.MesComutLocal	  	:= NOT IN_MesComutLocal_IO	    ; 
	MesDataExd.MesSwitchG		    := NOT IN_MesSwitchG_IO		    ; 
	MesDataExd.MesTest_Serv 	  	:= NOT IN_MesTest_Serv_IO 	    ; 
	MesDataExd.MesOpened_Sect 		:= NOT IN_MesOpened_Sect_IO 	; 
	MesDataExd.MesDefaulr_48VCC		:= NOT IN_MesDefaulr_48VCC_IO	; 

	ELSE
	MesDataExd.MesData.MesOpened	:=  IN_MesOpened_IO		    	; 
	MesDataExd.MesComutLocal	  	:=  IN_MesComutLocal_IO	    	; 
	MesDataExd.MesSwitchG		    :=  IN_MesSwitchG_IO			; 
	MesDataExd.MesTest_Serv 	  	:=  IN_MesTest_Serv_IO 	    	; 
	MesDataExd.MesOpened_Sect 		:=  IN_MesOpened_Sect_IO 		; 
	MesDataExd.MesDefaulr_48VCC		:=  IN_MesDefaulr_48VCC_IO		; 



	END_IF






	
MesDataExd.MesAlarmPwr		    := IN_MesAlarmPwr_IO ; 
MesDataExd.MesTripped			:= IN_MesTripped_IO ; 
MesDataExd.OUT_CmdClose		    := OUT_CmdClose_IO ; 
MesDataExd.OUT_CmdOpen		    := OUT_CmdOpen_IO ; 
MesDataExd.MesEarth			    := IN_MesEarth_IO ; 
//MesDataExd.MesOpened_Sect	    := SEL(ParamSectLigne.0, FALSE, A1_Sect.MesDataExd.MesData.MesOpened) ;
END_METHOD

METHOD M_Emulator
VAR_INPUT
END_VAR

TON_GTE_Default_Emul (IN:= IN_GTE_Default_Emul, PT := (ParamTP_Impulsion-T#100MS));
TON_OutputWait_Open(IN :=OUT_CmdOpen_IO, PT := (ParamTP_Impulsion-T#100MS));
TON_OutputWait_Close(IN :=OUT_CmdClose_IO, PT := (ParamTP_Impulsion-T#100MS));

R_TRIGOpen(CLK := TON_OutputWait_Open.Q);
R_TRIGClose(CLK := TON_OutputWait_Close.Q);    

RS_Emulate(SET := R_TRIGClose.Q OR CmdExternalClose_Emul , RESET1 := TON_GTE_Default_Emul.Q OR R_TRIGOpen.Q OR CmdExternalOpen_Emul ); 			// The Cell opens after receiving a open order or if receiving an external open ordre ( C13100 , .. ) 

IF ParamNC THEN 
	IN_MesOpened_IO 		:= RS_Emulate.Q1 ;  						
	IN_MesClosed_IO 		:= NOT RS_Emulate.Q1 ; 						
ELSE                                                                    
	IN_MesOpened_IO 		:= NOT RS_Emulate.Q1 ;  					
	IN_MesClosed_IO 		:= RS_Emulate.Q1 ; 							
END_IF
END_METHOD

METHOD M_Execute
VAR_INPUT
END_VAR

VAR

END_VAR
//MainMVCB avec etat de sectionneur de ligne
IF ParamSectLigne.0 THEN 
	A1_Sect.ParamNbFdbck := 1;
	A1_Sect.ParamNC := ParamSectLigne.1;
	A1_Sect.ParamClosedInput_Connected := TRUE ; 
	A1_Sect.M_Execute();
END_IF

// PERMANENT CONDITIONS //	
MesDataExd.MesData.MesCP_Open					:= IN_CmdOpen AND NOT IN_CmdReset;
MesDataExd.MesData.MesCP_Close				:= NOT MesDataExd.MesData.MesClosed AND IN_CmdClose AND NOT MesDataExd.MesData.MesAlarmCode.0 AND NOT MesDataExd.MesData.MesCP_Open AND NOT IN_CmdReset ;


SUPER^.M_Execute();
END_METHOD

METHOD M_OpenClose
//////////////////
// Manages Opening and Closing of the contactor
//////////////////

VAR 
	// Method local variables (reinitialized at each cycle) 

	
END_VAR
//AJOUT EXEPTION MAIN CIRCUIT BREAKER 
IF ParamSectLigne.0 THEN
	MesDataExd.MesData.MesCP_Close := MesDataExd.MesData.MesCP_Close AND NOT MesDataExd.MesOpened_Sect; // A1_Sect.IN_MesClosed_IO; //Check
END_IF
(*

Il peut y avoir 3 bobines :
 Bobine d'ouverture = on envoie un créneau pour fermer la cellule
 Bobine de fermeture = on envoie un créneau pour ouvrir la cellule
 Bobine à manque = si pas alimentée, la cellule ne peut pas rester fermée ni se fermer.
 Dans certaines cellules, il n'y a pas de bobine d'ouverture : il faut enlever l'alimentation de la bobine à manque pour que la cellule s'ouvre. 

*)

// ATTENTION : CODE NON TESTE ENCORE.
IF ParamUvCoil THEN
	RS_MaintainClose(set := MesDataExd.MesData.MesCP_Close OR NOT MesDataExd.MesData.MesCP_Open, RESET1 := MesDataExd.MesData.MesCP_Open);
	// je pourrais mettre que le Not CP_Open : il me permet d'être sûr que la bobine à manque est désactivée que quelques secondes
	OUT_CmdMaintainClose_IO := RS_MaintainClose.Q1;
END_IF


// Open Command
	ParamTP_Open(IN:= MesDataExd.MesData.MesCP_Open , PT:=ParamTP_Impulsion) ;
	OUT_CmdOpen_IO	 := ParamTP_Open.Q ;	// Impulsion that goes back to zero as soon as the state of the TP goes down. 

// Close Command
	ParamTP_Close(IN:= MesDataExd.MesData.MesCP_Close , PT:=ParamTP_Impulsion) ;
	OUT_CmdClose_IO	 := ParamTP_Close.Q ;   // Impulsion that goes back to zero as soon as the state of the TP goes down.
END_METHOD

METHOD M_StateManager
//////////////////
// Manages Contactor State
/////////////////

VAR 
	// Method local variables (reinitialized at each cycle) 
	
END_VAR
MesState := 0 ; 
IF MesOpened THEN		// If the cell seems opens and closed in the same time, we will consider it as opened. 
	
	MesState.0 := 1 ; 
MesDataExd.MesData.MesClosed := FALSE ; 
MesDataExd.MesData.MesOpened := TRUE ; 
ELSIF MesClosed THEN
	
	MesState.1 := 1 ; 
MesDataExd.MesData.MesClosed := TRUE ; 
MesDataExd.MesData.MesOpened := FALSE ; 
ELSE 
	MesState.0 := 1 ;		// if the cell seems neither opened and neither closed , we will consider it as opened. 
MesDataExd.MesData.MesClosed := FALSE ; 	
MesDataExd.MesData.MesOpened := TRUE ; 
END_IF
END_METHOD

END_FUNCTION_BLOCK

// ---- 01_Equipement_Library/Actuators/FB_CB_MeasureMVCB.TcPOU
FUNCTION_BLOCK FB_CB_MeasureMVCB EXTENDS FB_CB_Base
//////////////////
//  Motorized Circuit Breaker with telecommAND  Requires Open and Close impulsions.
//////////////////

VAR_INPUT PERSISTENT
	// Parameters of the Object (instance/model specific) 
	ParamTP_Impulsion	   : TIME := T#2S;			(* (s) 	 Config : Tempo for the start or stop command impulsion*)
	ParamFuseNC		       : BOOL;					(* (NA)	 False  : TRUE = Closed , True : TRUE = opened	*)
END_VAR

VAR_OUTPUT
	//Child objects
	
END_VAR

VAR_INPUT
	// I/O Inputs              
	IN_MesFuse_IO			: BOOL;
	IN_MesEarth_IO			: BOOL; 
	
	MesDataExd	: CB_MeasureMVCB_Sch ;
	
END_VAR

VAR
	//M_OPENCLOSE VARIABLES//	
		RsFuse				: RS ;
		
	//M_ALARMMANAGEMENT VARIABLES//

 
	//M_STATEMANAGER VARIABLES//
	
	// M_EXECUTE VARIABLES //
	
END_VAR

METHOD M_AlarmManagement
//////////////////
// Manages Contactor alarms and warnings
/////////////////

VAR 
	// Method local variables (reinitialized at each cycle) 
	FB_AlarmCodeManager			: FB_AlarmCodeManager ; 

	
END_VAR
// Check if command and measures are matching after tempo

TON_NotClosedAndNotOpened(IN:=  NOT MesClosed AND NOT MesOpened , PT := ParamTimeOut_Alarm) ; 
TON_ClosedAndOpened(IN:=MesClosed AND MesOpened, PT := ParamTimeOut_Alarm) ; 

RsFuse(Set:= MesDataExd.MesFuseBurned ,Reset1:=GVL_CFG.CmdClearFault_G OR IN_CmdReset);



// ALARM CODE //
	FB_AlarmCodeManager(
		bAlarm1			:= FALSE,										//
		bAlarm2			:= TON_NotClosedAndNotOpened.Q,					// Incoherent State measure (Not Opened and not Closed 
		bAlarm3 		:= TON_ClosedAndOpened.Q   , 					// Incoherent State measure (Opened and Closed )	
		bAlarm4			:= RsFuse.Q1,									// Fuse burned
		bAlarm5			:= FALSE, 										//  
		bAlarm6			:= FALSE, 										//
		bAlarm7			:= FALSE,                                       //
		bAlarm8			:= FALSE,                                       //
		bAlarm9			:= FALSE,                                       //
		bAlarm10		:= FALSE,                                       //
		bAlarm11		:= FALSE,                                       //
		bAlarm12		:= FALSE,                                       //
		bAlarm13		:= FALSE, 										//
		bAlarm14		:= FALSE, 										//
		bAlarm15		:= FALSE , 										// 
		wAlarmCode		=>MesDataExd.MesData.MesAlarmCode);

//WARNING CODE//
		FB_AlarmCodeManager(
		bAlarm1			:= FALSE , 										// 
		bAlarm2			:= FALSE  , 									// 
		bAlarm3 		:= FALSE,										// 
		bAlarm4			:= FALSE, 										// 
		bAlarm5			:= FALSE, 										//
		bAlarm6			:= MesDataExd.MesEarth, 						// The cell is connected to earth (earthing)
		bAlarm7			:= FALSE, 										//
		bAlarm8			:= FALSE,                                       //
		bAlarm9			:= FALSE,                                       //
		bAlarm10		:= FALSE,                                       //
		bAlarm11		:= FALSE,                                       //
		bAlarm12		:= FALSE,                                       //
		bAlarm13		:= FALSE,                                       //
		bAlarm14		:= FALSE,                                       //
		bAlarm15		:= FALSE, 										//
		wAlarmCode 		=>MesDataExd.MesData.MesWarningCode);

// EVENT CODE //
	FB_AlarmCodeManager(
		bAlarm1			:= FALSE, 										// 
		bAlarm2			:= FALSE, 										// 
		bAlarm3			:= MesOpened, 									// Opened Position
		bAlarm4			:= MesClosed, 									// Closed Position
		bAlarm5			:= IN_CmdReset, 								// Reset Command
		bAlarm6			:= FALSE, 										//
		bAlarm7			:= FALSE,                                       //
		bAlarm8			:= FALSE,                                       //
		bAlarm9			:= FALSE,                                       //
		bAlarm10		:= FALSE,                                       //
		bAlarm11		:= FALSE,                                       //
		bAlarm12		:= FALSE,                                       //
		bAlarm13		:= FALSE,                                       //
		bAlarm14		:= FALSE, 										//
		bAlarm15		:= FALSE, 										//
		wAlarmCode		=>MesDataExd.MesData.MesEventCode);
		
	// UPDATE STRUCTURE


		
	IF NOT ParamFuseNC THEN 
	MesDataExd.MesFuseBurned := NOT IN_MesFuse_IO;
	ELSE
	MesDataExd.MesFuseBurned := IN_MesFuse_IO;
	END_IF
	
MesDataExd.MesEarth	:= IN_MesEarth_IO ;
END_METHOD

METHOD M_Execute
VAR_INPUT
END_VAR

// PERMANENT CONDITIONS //	
MesDataExd.MesData.MesCP_Open					:= IN_CmdOpen AND NOT IN_CmdReset;
MesDataExd.MesData.MesCP_Close				:= NOT MesDataExd.MesData.MesClosed AND IN_CmdClose AND NOT MesDataExd.MesData.MesAlarmCode.0 AND NOT MesDataExd.MesData.MesCP_Open AND NOT IN_CmdReset ;


SUPER^.M_Execute();
END_METHOD

METHOD M_OpenClose
//////////////////
// Manages Opening and Closing of the contactor
//////////////////

VAR 
	// Method local variables (reinitialized at each cycle) 

	
END_VAR
END_METHOD

METHOD M_StateManager
//////////////////
// Manages Contactor State
/////////////////

VAR 
	// Method local variables (reinitialized at each cycle) 
	
END_VAR
MesState := 0 ; 
IF MesOpened THEN		// If the cell seems opens and closed in the same time, we will consider it as opened. 
	
	MesState.0 := 1 ; 
MesDataExd.MesData.MesClosed := FALSE ; 
MesDataExd.MesData.MesOpened := TRUE ; 
ELSIF MesClosed THEN
	
	MesState.1 := 1 ; 
MesDataExd.MesData.MesClosed := TRUE ; 
MesDataExd.MesData.MesOpened := FALSE ; 
ELSE 
	MesState.0 := 1 ;		// if the cell seems neither opened and neither closed , we will consider it as opened. 
MesDataExd.MesData.MesClosed := FALSE ; 	
MesDataExd.MesData.MesOpened := TRUE ; 
END_IF
END_METHOD

END_FUNCTION_BLOCK

// ---- 01_Equipement_Library/Actuators/FB_CB_FeederMVCB.TcPOU
FUNCTION_BLOCK FB_CB_FeederMVCB EXTENDS FB_CB_Base
//////////////////
//  Motorized Circuit Breaker with telecommAND   Requires Open and Close impulsions.
//////////////////

VAR_INPUT PERSISTENT
	// Parameters of the Object (instance/model specific) 
	ParamTP_Impulsion		    : TIME 		:= T#2S;	(* (s) Config : Tempo for the start or stop command impulsion*)
	ParamComutNc			    : BOOL;					(* (NA) Local selector in normally closed. NC >> True = Selector in local. *)
	ParamSectLigne			    : BYTE      :=1;		(* (NA) Monitoring du sectionneur de ligne de la MainMVCB.0 = TRUE := Monitoré .1 = TRUE Close is connected*)

END_VAR
VAR_INPUT
	A1_Sect				       : FB_CB_MVSwitch;

// Fire Ditection 	
	IN_FireDetection			: BOOL ;				// Set to TRUE if there is a fire in the PTR

// I/O Inputs              
	IN_MesAlarmPwr_IO		   : BOOL ;	              // (NA)[P,H,B] Remote control Power supply Error IO  	
	IN_MesTripped_IO		   : BOOL ; 	          // Tripped position of the CB Must Ack To switch in again
	IN_MesComutLocal_IO		   : BOOL ;	 	 		 // True if cell is in local position 
	IN_MesEarth_IO 			   : BOOL ; 	

	MesDataExd					: CB_FeederMVCB_Sch ; 
		
END_VAR

VAR_OUTPUT
	//Child objects
	OUT_CmdOpen_IO	           : BOOL ; 	          // (NA) Physical I/O Open Command IO
	OUT_CmdClose_IO			   : BOOL ; 	          // (NA) Physical I/O Close Command IO
	
END_VAR


VAR
	//M_OPENCLOSE VARIABLES//

	//M_OPENCLOSE VARIABLES//	
	ParamTP_Open	 			: TP ;				(* (NA) Temporisation for Open pulse Command*)
	ParamTP_Close 				: TP ;				(* (NA) Temporisation for Close pulse Command	*)
		
END_VAR

METHOD M_AlarmManagement
//////////////////
// Manages Contactor alarms and warnings
/////////////////

VAR 
	// Method local variables (reinitialized at each cycle) 
	FB_AlarmCodeManager			: FB_AlarmCodeManager ; 
	bSectLigne					: BOOL;
END_VAR
VAR_INPUT
	
END_VAR
// Check if command and measures are matching after tempo
FB_CheckCommand	(T:= ParamTimeOut_Close, bCmd:=OUT_CmdClose_IO , bMes := MesDataExd.MesData.MesClosed , bImpulsion := FALSE , bReset := CmdClearFault_G OR OUT_CmdClose_IO) ; 
FB_CheckCommand2(T:= ParamTimeOut_Open , bCmd:= OUT_CmdOpen_IO , bMes :=NOT MesDataExd.MesData.MesClosed , bImpulsion := FALSE , bReset := CmdClearFault_G OR OUT_CmdOpen_IO) ; 

TON_NotClosedAndNotOpened(IN:=  NOT MesClosed AND NOT MesOpened , PT := ParamTimeOut_Alarm) ; 
TON_ClosedAndOpened(IN:=MesClosed AND MesOpened, PT := ParamTimeOut_Alarm) ; 

// ALARM CODE //
	FB_AlarmCodeManager(
		bAlarm1			:= MesDataExd.MesTripped,						// CB is tripped
		bAlarm2			:= TON_NotClosedAndNotOpened.Q,					// Incoherent State measure (Not Opened and not Closed)
		bAlarm3 		:= TON_ClosedAndOpened.Q   , 					// Incoherent State measure (Opened and Closed)	
		bAlarm4			:= FB_CheckCommAND.bWarning , 					// Close command failed
		bAlarm5			:= FB_CheckCommand2.bWarning  , 				// Open Command failed
		bAlarm6			:= FALSE,                                   	//
		bAlarm7			:= FALSE,                                   	//
		bAlarm8			:= FALSE,                                   	//
		bAlarm9			:= FALSE,                                   	//
		bAlarm10		:= FALSE,                                   	//
		bAlarm11		:= FALSE,                                   	//
		bAlarm12		:= FALSE,                                   	//
		bAlarm13		:= FALSE,                                   	//
		bAlarm14		:= FALSE,                                   	//
		bAlarm15		:= FALSE , 										//
		wAlarmCode		=>MesDataExd.MesData.MesAlarmCode);

		
	bSectLigne := SEL(ParamSectLigne.0 ,FALSE , NOT A1_Sect.MesDataExd.MesData.MesClosed);
//WARNING CODE//

// Attention une alarm doit être mise en commentaire de la manière suivante (* *), l'utilisation du // pose pb sur Bazefield 

		FB_AlarmCodeManager(
		bAlarm1			:= FALSE,										//
		bAlarm2			:= FALSE,										//
		bAlarm3 		:= FALSE,										// 
		bAlarm4			:= MesDataExd.MesAlarmPwr, 						// Power supply fault
		bAlarm5			:= MesDataExd.MesComutLocal, 					// Commutator in local mode 
		bAlarm6			:= MesDataExd.MesEarth, 						// The cell is connected to earth (earthing)
		bAlarm7			:= bSectLigne,	// Line connector is opened (sectionneur)
		bAlarm8			:= FALSE, 										//
		bAlarm9			:= FALSE,                                       //
		bAlarm10		:= FALSE,                                       //
		bAlarm11		:= FALSE,                                       //
		bAlarm12		:= FALSE,                                       //
		bAlarm13		:= FALSE,                                       //
		bAlarm14		:= FALSE,                                       //
		bAlarm15		:= FALSE, 										//
		wAlarmCode 		=>MesDataExd.MesData.MesWarningCode);

// EVENT CODE //
	FB_AlarmCodeManager(
		bAlarm1			:= OUT_CmdOpen_IO, 								// Open Command
		bAlarm2			:= OUT_CmdClose_IO, 							// Close Command
		bAlarm3			:= MesOpened, 									// Opened Position
		bAlarm4			:= MesClosed, 									// Closed Position
		bAlarm5			:= IN_CmdReset, 								// Reset command
		bAlarm6			:= FALSE, 										//
		bAlarm7			:= FALSE,                   					//
		bAlarm8			:= FALSE,                   					//
		bAlarm9			:= FALSE,                   					//
		bAlarm10		:= FALSE,                   					//
		bAlarm11		:= FALSE,                   					//
		bAlarm12		:= FALSE,                   					//
		bAlarm13		:= FALSE, 										//
		bAlarm14		:= FALSE,                   					//
		bAlarm15		:= FALSE,                   					//
		wAlarmCode		=>MesDataExd.MesData.MesEventCode);   
                                           
	// UPDATE STRUCTURE	
	IF ParamComutNc THEN
	MesDataExd.MesComutLocal	:= NOT IN_MesComutLocal_IO ; 
	ELSE
	MesDataExd.MesComutLocal	:= IN_MesComutLocal_IO ; 
	END_IF
	
MesDataExd.MesAlarmPwr		    := IN_MesAlarmPwr_IO ; 
MesDataExd.MesTripped			:= IN_MesTripped_IO ; 
MesDataExd.OUT_CmdClose		    := OUT_CmdClose_IO ; 
MesDataExd.OUT_CmdOpen		    := OUT_CmdOpen_IO ; 
MesDataExd.MesEarth			    := IN_MesEarth_IO ; 
MesDataExd.MesOpened_Sect	        := SEL(ParamSectLigne.0 , FALSE  , NOT A1_Sect.MesDataExd.MesData.MesClosed ) ; 
	
	//MesDataExd	    := MesDataExd.MesData.;
END_METHOD

METHOD M_Emulator
VAR_INPUT
END_VAR
TON_OutputWait_Open(IN :=OUT_CmdOpen_IO, PT := ParamTP_Impulsion-T#100MS);
TON_OutputWait_Close(IN :=OUT_CmdClose_IO, PT := ParamTP_Impulsion-T#100MS);

R_TRIGOpen(CLK := TON_OutputWait_Open.Q);
R_TRIGClose(CLK := TON_OutputWait_Close.Q);    

RS_Emulate(SET := R_TRIGClose.Q OR CmdExternalClose_Emul , RESET1 := R_TRIGOpen.Q OR CmdExternalOpen_Emul ); 			// The Cell opens after receiving a open order or if receiving an external open ordre ( C13100 , .. ) 

IF ParamNC THEN 
	IN_MesOpened_IO 		:= RS_Emulate.Q1 ;  						
	IN_MesClosed_IO 		:= NOT RS_Emulate.Q1 ; 						
ELSE                                                                    
	IN_MesOpened_IO 		:= NOT RS_Emulate.Q1 ;  					
	IN_MesClosed_IO 		:= RS_Emulate.Q1 ; 							
END_IF
END_METHOD

METHOD M_Execute
VAR_INPUT
END_VAR

VAR

END_VAR
//MainMVCB avec etat de sectionneur de ligne
IF ParamSectLigne.0 THEN 
	A1_Sect.ParamNbFdbck := 1;
	A1_Sect.ParamClosedInput_Connected := TRUE ; 
	A1_Sect.M_Execute();
END_IF

// PERMANENT CONDITIONS //	
MesDataExd.MesData.MesCP_Open				:= IN_FireDetection OR (IN_CmdOpen AND NOT IN_CmdReset_L);
MesDataExd.MesData.MesCP_Close				:= NOT IN_FireDetection AND NOT MesDataExd.MesData.MesClosed AND IN_CmdClose AND NOT MesDataExd.MesData.MesAlarmCode.0 AND NOT MesDataExd.MesData.MesCP_Open AND NOT IN_CmdReset_L  ;



SUPER^.M_Execute();
END_METHOD

METHOD M_OpenClose
//////////////////
// Manages Opening and Closing of the contactor
//////////////////

VAR 
	// Method local variables (reinitialized at each cycle) 

	
END_VAR
//AJOUT EXEPTION MAIN CIRCUIT BREAKER 
IF ParamSectLigne.0 THEN
MesDataExd.MesData.MesCP_Close := MesDataExd.MesData.MesCP_Close AND A1_Sect.IN_MesClosed_IO; //Check
END_IF

// Open Command
ParamTP_Open(IN:= MesDataExd.MesData.MesCP_Open , PT:=ParamTP_Impulsion) ;
OUT_CmdOpen_IO	 := ParamTP_Open.Q ;                               			 // Impulsion that goes back to zero as soon as the state of the TP goes down. 

// Close Command
ParamTP_Close(IN:= MesDataExd.MesData.MesCP_Close , PT:=ParamTP_Impulsion) ;
OUT_CmdClose_IO	 := ParamTP_Close.Q ;                          			 // Impulsion that goes back to zero as soon as the state of the TP goes down.
END_METHOD

METHOD M_StateManager
//////////////////
// Manages Contactor State
/////////////////

VAR 
	// Method local variables (reinitialized at each cycle) 
	
END_VAR
MesState := 0 ; 
IF MesOpened THEN		// If the cell seems opens and closed in the same time, we will consider it as opened. 
	
	MesState.0 := 1 ; 
MesDataExd.MesData.MesClosed := FALSE ; 
MesDataExd.MesData.MesOpened := TRUE ; 
ELSIF MesClosed THEN
	
	MesState.1 := 1 ; 
MesDataExd.MesData.MesClosed := TRUE ; 
MesDataExd.MesData.MesOpened := FALSE ; 
ELSE 
	MesState.0 := 1 ;		// if the cell seems neither opened and neither closed , we will consider it as opened. 
MesDataExd.MesData.MesClosed := FALSE ; 	
MesDataExd.MesData.MesOpened := TRUE ; 
END_IF
END_METHOD

END_FUNCTION_BLOCK

// ---- 01_Equipement_Library/Actuators/FB_CB_Switch.TcPOU
FUNCTION_BLOCK FB_CB_Switch EXTENDS FB_CB_Base
//////////////////
//  Motorized Circuit Breaker with telecommAND   Requires Open and Close impulsions.
//////////////////

VAR_INPUT PERSISTENT
	// Parameters of the Object (instance/model specific) 
	ParamTP_Impulsion		    : TIME 		:= T#2S;	(* (s) Config : Tempo for the start or stop command impulsion*)
END_VAR

VAR_INPUT
	

